(* Logix 5000 project; controller reports 1756-L63 rev 20.11; software revision 20.04; part 5 of 52 *)

        [413].time.Second := 59, [414].log_data[0].min := 1.0, [414].log_data[0].max := 1.0, [414].log_data[0].total := 900.0, [414].log_data[0].time := 900.0, [414].log_data[0].minminute := 45, [414].log_data[0].maxminute := 45, [414].log_data[0].valid := 1, [414].log_data[1].valid := 1, [414].log_data[2].valid := 1, [414].log_data[3].valid := 1, [414].log_data[4].valid := 1, [414].log_data[5].valid := 1, [414].log_data[6].valid := 1, [414].log_data[7].valid := 1, [414].log_data[8].valid := 1, [414].log_data[9].valid := 1, [414].log_data[10].valid := 1, [414].log_data[11].valid := 1, [414].log_data[12].valid := 1, [414].log_data[13].valid := 1, [414].log_data[14].valid := 1, [414].log_data[15].valid := 1, [414].log_data[16].valid := 1, [414].log_data[17].valid := 1, [414].log_data[18].valid := 1, [414].log_data[19].valid := 1, [414].time.Year := 2023, [414].time.Month := 1, [414].time.Day := 11, [414].time.Hour := 23, [414].time.Minute := 59, [414].time.Second := 59, [415].log_data[0].min := 1.0, [415].log_data[0].max := 1.0, [415].log_data[0].total := 900.0, [415].log_data[0].time := 900.0, [415].log_data[0].valid := 1, [415].log_data[1].valid := 1, [415].log_data[2].valid := 1, [415].log_data[3].valid := 1, [415].log_data[4].valid := 1, [415].log_data[5].valid := 1, [415].log_data[6].valid := 1, [415].log_data[7].valid := 1, [415].log_data[8].valid := 1, [415].log_data[9].valid := 1, [415].log_data[10].valid := 1, [415].log_data[11].valid := 1, [415].log_data[12].valid := 1, [415].log_data[13].valid := 1, [415].log_data[14].valid := 1, [415].log_data[15].valid := 1, [415].log_data[16].valid := 1, [415].log_data[17].valid := 1, [415].log_data[18].valid := 1, [415].log_data[19].valid := 1, [415].time.Year := 2023, [415].time.Month := 1, [415].time.Day := 12,
        [415].time.Minute := 14, [415].time.Second := 59, [416].log_data[0].min := 1.0, [416].log_data[0].max := 1.0, [416].log_data[0].total := 900.0, [416].log_data[0].time := 900.0, [416].log_data[0].minminute := 15, [416].log_data[0].maxminute := 15, [416].log_data[0].valid := 1, [416].log_data[1].valid := 1, [416].log_data[2].valid := 1, [416].log_data[3].valid := 1, [416].log_data[4].valid := 1, [416].log_data[5].valid := 1, [416].log_data[6].valid := 1, [416].log_data[7].valid := 1, [416].log_data[8].valid := 1, [416].log_data[9].valid := 1, [416].log_data[10].valid := 1, [416].log_data[11].valid := 1, [416].log_data[12].valid := 1, [416].log_data[13].valid := 1, [416].log_data[14].valid := 1, [416].log_data[15].valid := 1, [416].log_data[16].valid := 1, [416].log_data[17].valid := 1, [416].log_data[18].valid := 1, [416].log_data[19].valid := 1, [416].time.Year := 2023, [416].time.Month := 1, [416].time.Day := 12, [416].time.Minute := 29, [416].time.Second := 59, [417].log_data[0].min := 1.0, [417].log_data[0].max := 1.0, [417].log_data[0].total := 900.0, [417].log_data[0].time := 900.0, [417].log_data[0].minminute := 30, [417].log_data[0].maxminute := 30, [417].log_data[0].valid := 1, [417].log_data[1].valid := 1, [417].log_data[2].valid := 1, [417].log_data[3].valid := 1, [417].log_data[4].valid := 1, [417].log_data[5].valid := 1, [417].log_data[6].valid := 1, [417].log_data[7].valid := 1, [417].log_data[8].valid := 1, [417].log_data[9].valid := 1, [417].log_data[10].valid := 1, [417].log_data[11].valid := 1, [417].log_data[12].valid := 1, [417].log_data[13].valid := 1, [417].log_data[14].valid := 1, [417].log_data[15].valid := 1, [417].log_data[16].valid := 1, [417].log_data[17].valid := 1, [417].log_data[18].valid := 1, [417].log_data[19].valid := 1, [417].time.Year := 2023,
        [417].time.Month := 1, [417].time.Day := 12, [417].time.Minute := 44, [417].time.Second := 59, [418].log_data[0].min := 1.0, [418].log_data[0].max := 1.0, [418].log_data[0].total := 900.0, [418].log_data[0].time := 900.0, [418].log_data[0].minminute := 45, [418].log_data[0].maxminute := 45, [418].log_data[0].valid := 1, [418].log_data[1].valid := 1, [418].log_data[2].valid := 1, [418].log_data[3].valid := 1, [418].log_data[4].valid := 1, [418].log_data[5].valid := 1, [418].log_data[6].valid := 1, [418].log_data[7].valid := 1, [418].log_data[8].valid := 1, [418].log_data[9].valid := 1, [418].log_data[10].valid := 1, [418].log_data[11].valid := 1, [418].log_data[12].valid := 1, [418].log_data[13].valid := 1, [418].log_data[14].valid := 1, [418].log_data[15].valid := 1, [418].log_data[16].valid := 1, [418].log_data[17].valid := 1, [418].log_data[18].valid := 1, [418].log_data[19].valid := 1, [418].time.Year := 2023, [418].time.Month := 1, [418].time.Day := 12, [418].time.Minute := 59, [418].time.Second := 59, [419].log_data[0].min := 1.0, [419].log_data[0].max := 1.0, [419].log_data[0].total := 899.5, [419].log_data[0].time := 899.5, [419].log_data[0].valid := 1, [419].log_data[1].valid := 1, [419].log_data[2].valid := 1, [419].log_data[3].valid := 1, [419].log_data[4].valid := 1, [419].log_data[5].valid := 1, [419].log_data[6].valid := 1, [419].log_data[7].valid := 1, [419].log_data[8].valid := 1, [419].log_data[9].valid := 1, [419].log_data[10].valid := 1, [419].log_data[11].valid := 1, [419].log_data[12].valid := 1, [419].log_data[13].valid := 1, [419].log_data[14].valid := 1, [419].log_data[15].valid := 1, [419].log_data[16].valid := 1, [419].log_data[17].valid := 1, [419].log_data[18].valid := 1, [419].log_data[19].valid := 1, [419].time.Year := 2023,
        [419].time.Month := 1, [419].time.Day := 12, [419].time.Hour := 1, [419].time.Minute := 14, [419].time.Second := 59, [420].log_data[0].min := 1.0, [420].log_data[0].max := 1.0, [420].log_data[0].total := 900.0, [420].log_data[0].time := 900.0, [420].log_data[0].minminute := 15, [420].log_data[0].maxminute := 15, [420].log_data[0].valid := 1, [420].log_data[1].valid := 1, [420].log_data[2].valid := 1, [420].log_data[3].valid := 1, [420].log_data[4].valid := 1, [420].log_data[5].valid := 1, [420].log_data[6].valid := 1, [420].log_data[7].valid := 1, [420].log_data[8].valid := 1, [420].log_data[9].valid := 1, [420].log_data[10].valid := 1, [420].log_data[11].valid := 1, [420].log_data[12].valid := 1, [420].log_data[13].valid := 1, [420].log_data[14].valid := 1, [420].log_data[15].valid := 1, [420].log_data[16].valid := 1, [420].log_data[17].valid := 1, [420].log_data[18].valid := 1, [420].log_data[19].valid := 1, [420].time.Year := 2023, [420].time.Month := 1, [420].time.Day := 12, [420].time.Hour := 1, [420].time.Minute := 29, [420].time.Second := 59, [421].log_data[0].min := 1.0, [421].log_data[0].max := 1.0, [421].log_data[0].total := 900.0, [421].log_data[0].time := 900.0, [421].log_data[0].minminute := 30, [421].log_data[0].maxminute := 30, [421].log_data[0].valid := 1, [421].log_data[1].valid := 1, [421].log_data[2].valid := 1, [421].log_data[3].valid := 1, [421].log_data[4].valid := 1, [421].log_data[5].valid := 1, [421].log_data[6].valid := 1, [421].log_data[7].valid := 1, [421].log_data[8].valid := 1, [421].log_data[9].valid := 1, [421].log_data[10].valid := 1, [421].log_data[11].valid := 1, [421].log_data[12].valid := 1, [421].log_data[13].valid := 1, [421].log_data[14].valid := 1, [421].log_data[15].valid := 1, [421].log_data[16].valid := 1,
        [421].log_data[17].valid := 1, [421].log_data[18].valid := 1, [421].log_data[19].valid := 1, [421].time.Year := 2023, [421].time.Month := 1, [421].time.Day := 12, [421].time.Hour := 1, [421].time.Minute := 44, [421].time.Second := 59, [422].log_data[0].min := 1.0, [422].log_data[0].max := 1.0, [422].log_data[0].total := 900.0, [422].log_data[0].time := 900.0, [422].log_data[0].minminute := 45, [422].log_data[0].maxminute := 45, [422].log_data[0].valid := 1, [422].log_data[1].valid := 1, [422].log_data[2].valid := 1, [422].log_data[3].valid := 1, [422].log_data[4].valid := 1, [422].log_data[5].valid := 1, [422].log_data[6].valid := 1, [422].log_data[7].valid := 1, [422].log_data[8].valid := 1, [422].log_data[9].valid := 1, [422].log_data[10].valid := 1, [422].log_data[11].valid := 1, [422].log_data[12].valid := 1, [422].log_data[13].valid := 1, [422].log_data[14].valid := 1, [422].log_data[15].valid := 1, [422].log_data[16].valid := 1, [422].log_data[17].valid := 1, [422].log_data[18].valid := 1, [422].log_data[19].valid := 1, [422].time.Year := 2023, [422].time.Month := 1, [422].time.Day := 12, [422].time.Hour := 1, [422].time.Minute := 59, [422].time.Second := 59, [423].log_data[0].min := 1.0, [423].log_data[0].max := 1.0, [423].log_data[0].total := 900.0, [423].log_data[0].time := 900.0, [423].log_data[0].valid := 1, [423].log_data[1].valid := 1, [423].log_data[2].valid := 1, [423].log_data[3].valid := 1, [423].log_data[4].valid := 1, [423].log_data[5].valid := 1, [423].log_data[6].valid := 1, [423].log_data[7].valid := 1, [423].log_data[8].valid := 1, [423].log_data[9].valid := 1, [423].log_data[10].valid := 1, [423].log_data[11].valid := 1, [423].log_data[12].valid := 1, [423].log_data[13].valid := 1, [423].log_data[14].valid := 1,
        [423].log_data[15].valid := 1, [423].log_data[16].valid := 1, [423].log_data[17].valid := 1, [423].log_data[18].valid := 1, [423].log_data[19].valid := 1, [423].time.Year := 2023, [423].time.Month := 1, [423].time.Day := 12, [423].time.Hour := 2, [423].time.Minute := 14, [423].time.Second := 59, [424].log_data[0].min := 1.0, [424].log_data[0].max := 1.0, [424].log_data[0].total := 900.0, [424].log_data[0].time := 900.0, [424].log_data[0].minminute := 15, [424].log_data[0].maxminute := 15, [424].log_data[0].valid := 1, [424].log_data[1].valid := 1, [424].log_data[2].valid := 1, [424].log_data[3].valid := 1, [424].log_data[4].valid := 1, [424].log_data[5].valid := 1, [424].log_data[6].valid := 1, [424].log_data[7].valid := 1, [424].log_data[8].valid := 1, [424].log_data[9].valid := 1, [424].log_data[10].valid := 1, [424].log_data[11].valid := 1, [424].log_data[12].valid := 1, [424].log_data[13].valid := 1, [424].log_data[14].valid := 1, [424].log_data[15].valid := 1, [424].log_data[16].valid := 1, [424].log_data[17].valid := 1, [424].log_data[18].valid := 1, [424].log_data[19].valid := 1, [424].time.Year := 2023, [424].time.Month := 1, [424].time.Day := 12, [424].time.Hour := 2, [424].time.Minute := 29, [424].time.Second := 59, [425].log_data[0].min := 1.0, [425].log_data[0].max := 1.0, [425].log_data[0].total := 900.0, [425].log_data[0].time := 900.0, [425].log_data[0].minminute := 30, [425].log_data[0].maxminute := 30, [425].log_data[0].valid := 1, [425].log_data[1].valid := 1, [425].log_data[2].valid := 1, [425].log_data[3].valid := 1, [425].log_data[4].valid := 1, [425].log_data[5].valid := 1, [425].log_data[6].valid := 1, [425].log_data[7].valid := 1, [425].log_data[8].valid := 1, [425].log_data[9].valid := 1, [425].log_data[10].valid := 1,
        [425].log_data[11].valid := 1, [425].log_data[12].valid := 1, [425].log_data[13].valid := 1, [425].log_data[14].valid := 1, [425].log_data[15].valid := 1, [425].log_data[16].valid := 1, [425].log_data[17].valid := 1, [425].log_data[18].valid := 1, [425].log_data[19].valid := 1, [425].time.Year := 2023, [425].time.Month := 1, [425].time.Day := 12, [425].time.Hour := 2, [425].time.Minute := 44, [425].time.Second := 59, [426].log_data[0].min := 1.0, [426].log_data[0].max := 1.0, [426].log_data[0].total := 900.0, [426].log_data[0].time := 900.0, [426].log_data[0].minminute := 45, [426].log_data[0].maxminute := 45, [426].log_data[0].valid := 1, [426].log_data[1].valid := 1, [426].log_data[2].valid := 1, [426].log_data[3].valid := 1, [426].log_data[4].valid := 1, [426].log_data[5].valid := 1, [426].log_data[6].valid := 1, [426].log_data[7].valid := 1, [426].log_data[8].valid := 1, [426].log_data[9].valid := 1, [426].log_data[10].valid := 1, [426].log_data[11].valid := 1, [426].log_data[12].valid := 1, [426].log_data[13].valid := 1, [426].log_data[14].valid := 1, [426].log_data[15].valid := 1, [426].log_data[16].valid := 1, [426].log_data[17].valid := 1, [426].log_data[18].valid := 1, [426].log_data[19].valid := 1, [426].time.Year := 2023, [426].time.Month := 1, [426].time.Day := 12, [426].time.Hour := 2, [426].time.Minute := 59, [426].time.Second := 59, [427].log_data[0].min := 1.0, [427].log_data[0].max := 1.0, [427].log_data[0].total := 900.0, [427].log_data[0].time := 900.0, [427].log_data[0].valid := 1, [427].log_data[1].valid := 1, [427].log_data[2].valid := 1, [427].log_data[3].valid := 1, [427].log_data[4].valid := 1, [427].log_data[5].valid := 1, [427].log_data[6].valid := 1, [427].log_data[7].valid := 1, [427].log_data[8].valid := 1,
        [427].log_data[9].valid := 1, [427].log_data[10].valid := 1, [427].log_data[11].valid := 1, [427].log_data[12].valid := 1, [427].log_data[13].valid := 1, [427].log_data[14].valid := 1, [427].log_data[15].valid := 1, [427].log_data[16].valid := 1, [427].log_data[17].valid := 1, [427].log_data[18].valid := 1, [427].log_data[19].valid := 1, [427].time.Year := 2023, [427].time.Month := 1, [427].time.Day := 12, [427].time.Hour := 3, [427].time.Minute := 14, [427].time.Second := 59, [428].log_data[0].min := 1.0, [428].log_data[0].max := 1.0, [428].log_data[0].total := 900.0, [428].log_data[0].time := 900.0, [428].log_data[0].minminute := 15, [428].log_data[0].maxminute := 15, [428].log_data[0].valid := 1, [428].log_data[1].valid := 1, [428].log_data[2].valid := 1, [428].log_data[3].valid := 1, [428].log_data[4].valid := 1, [428].log_data[5].valid := 1, [428].log_data[6].valid := 1, [428].log_data[7].valid := 1, [428].log_data[8].valid := 1, [428].log_data[9].valid := 1, [428].log_data[10].valid := 1, [428].log_data[11].valid := 1, [428].log_data[12].valid := 1, [428].log_data[13].valid := 1, [428].log_data[14].valid := 1, [428].log_data[15].valid := 1, [428].log_data[16].valid := 1, [428].log_data[17].valid := 1, [428].log_data[18].valid := 1, [428].log_data[19].valid := 1, [428].time.Year := 2023, [428].time.Month := 1, [428].time.Day := 12, [428].time.Hour := 3, [428].time.Minute := 29, [428].time.Second := 59, [429].log_data[0].min := 1.0, [429].log_data[0].max := 1.0, [429].log_data[0].total := 900.0, [429].log_data[0].time := 900.0, [429].log_data[0].minminute := 30, [429].log_data[0].maxminute := 30, [429].log_data[0].valid := 1, [429].log_data[1].valid := 1, [429].log_data[2].valid := 1, [429].log_data[3].valid := 1, [429].log_data[4].valid := 1,
        [429].log_data[5].valid := 1, [429].log_data[6].valid := 1, [429].log_data[7].valid := 1, [429].log_data[8].valid := 1, [429].log_data[9].valid := 1, [429].log_data[10].valid := 1, [429].log_data[11].valid := 1, [429].log_data[12].valid := 1, [429].log_data[13].valid := 1, [429].log_data[14].valid := 1, [429].log_data[15].valid := 1, [429].log_data[16].valid := 1, [429].log_data[17].valid := 1, [429].log_data[18].valid := 1, [429].log_data[19].valid := 1, [429].time.Year := 2023, [429].time.Month := 1, [429].time.Day := 12, [429].time.Hour := 3, [429].time.Minute := 44, [429].time.Second := 59, [430].log_data[0].min := 1.0, [430].log_data[0].max := 1.0, [430].log_data[0].total := 900.0, [430].log_data[0].time := 900.0, [430].log_data[0].minminute := 45, [430].log_data[0].maxminute := 45, [430].log_data[0].valid := 1, [430].log_data[1].valid := 1, [430].log_data[2].valid := 1, [430].log_data[3].valid := 1, [430].log_data[4].valid := 1, [430].log_data[5].valid := 1, [430].log_data[6].valid := 1, [430].log_data[7].valid := 1, [430].log_data[8].valid := 1, [430].log_data[9].valid := 1, [430].log_data[10].valid := 1, [430].log_data[11].valid := 1, [430].log_data[12].valid := 1, [430].log_data[13].valid := 1, [430].log_data[14].valid := 1, [430].log_data[15].valid := 1, [430].log_data[16].valid := 1, [430].log_data[17].valid := 1, [430].log_data[18].valid := 1, [430].log_data[19].valid := 1, [430].time.Year := 2023, [430].time.Month := 1, [430].time.Day := 12, [430].time.Hour := 3, [430].time.Minute := 59, [430].time.Second := 59, [431].log_data[0].min := 1.0, [431].log_data[0].max := 1.0, [431].log_data[0].total := 900.0, [431].log_data[0].time := 900.0, [431].log_data[0].valid := 1, [431].log_data[1].valid := 1, [431].log_data[2].valid := 1,
        [431].log_data[3].valid := 1, [431].log_data[4].valid := 1, [431].log_data[5].valid := 1, [431].log_data[6].valid := 1, [431].log_data[7].valid := 1, [431].log_data[8].valid := 1, [431].log_data[9].valid := 1, [431].log_data[10].valid := 1, [431].log_data[11].valid := 1, [431].log_data[12].valid := 1, [431].log_data[13].valid := 1, [431].log_data[14].valid := 1, [431].log_data[15].valid := 1, [431].log_data[16].valid := 1, [431].log_data[17].valid := 1, [431].log_data[18].valid := 1, [431].log_data[19].valid := 1, [431].time.Year := 2023, [431].time.Month := 1, [431].time.Day := 12, [431].time.Hour := 4, [431].time.Minute := 14, [431].time.Second := 59, [432].log_data[0].min := 1.0, [432].log_data[0].max := 1.0, [432].log_data[0].total := 900.0, [432].log_data[0].time := 900.0, [432].log_data[0].minminute := 15, [432].log_data[0].maxminute := 15, [432].log_data[0].valid := 1, [432].log_data[1].valid := 1, [432].log_data[2].valid := 1, [432].log_data[3].valid := 1, [432].log_data[4].valid := 1, [432].log_data[5].valid := 1, [432].log_data[6].valid := 1, [432].log_data[7].valid := 1, [432].log_data[8].valid := 1, [432].log_data[9].valid := 1, [432].log_data[10].valid := 1, [432].log_data[11].valid := 1, [432].log_data[12].valid := 1, [432].log_data[13].valid := 1, [432].log_data[14].valid := 1, [432].log_data[15].valid := 1, [432].log_data[16].valid := 1, [432].log_data[17].valid := 1, [432].log_data[18].valid := 1, [432].log_data[19].valid := 1, [432].time.Year := 2023, [432].time.Month := 1, [432].time.Day := 12, [432].time.Hour := 4, [432].time.Minute := 29, [432].time.Second := 59, [433].log_data[0].min := 1.0, [433].log_data[0].max := 1.0, [433].log_data[0].total := 900.0, [433].log_data[0].time := 900.0, [433].log_data[0].minminute := 30,
        [433].log_data[0].maxminute := 30, [433].log_data[0].valid := 1, [433].log_data[1].valid := 1, [433].log_data[2].valid := 1, [433].log_data[3].valid := 1, [433].log_data[4].valid := 1, [433].log_data[5].valid := 1, [433].log_data[6].valid := 1, [433].log_data[7].valid := 1, [433].log_data[8].valid := 1, [433].log_data[9].valid := 1, [433].log_data[10].valid := 1, [433].log_data[11].valid := 1, [433].log_data[12].valid := 1, [433].log_data[13].valid := 1, [433].log_data[14].valid := 1, [433].log_data[15].valid := 1, [433].log_data[16].valid := 1, [433].log_data[17].valid := 1, [433].log_data[18].valid := 1, [433].log_data[19].valid := 1, [433].time.Year := 2023, [433].time.Month := 1, [433].time.Day := 12, [433].time.Hour := 4, [433].time.Minute := 44, [433].time.Second := 59, [434].log_data[0].min := 1.0, [434].log_data[0].max := 1.0, [434].log_data[0].total := 900.0, [434].log_data[0].time := 900.0, [434].log_data[0].minminute := 45, [434].log_data[0].maxminute := 45, [434].log_data[0].valid := 1, [434].log_data[1].valid := 1, [434].log_data[2].valid := 1, [434].log_data[3].valid := 1, [434].log_data[4].valid := 1, [434].log_data[5].valid := 1, [434].log_data[6].valid := 1, [434].log_data[7].valid := 1, [434].log_data[8].valid := 1, [434].log_data[9].valid := 1, [434].log_data[10].valid := 1, [434].log_data[11].valid := 1, [434].log_data[12].valid := 1, [434].log_data[13].valid := 1, [434].log_data[14].valid := 1, [434].log_data[15].valid := 1, [434].log_data[16].valid := 1, [434].log_data[17].valid := 1, [434].log_data[18].valid := 1, [434].log_data[19].valid := 1, [434].time.Year := 2023, [434].time.Month := 1, [434].time.Day := 12, [434].time.Hour := 4, [434].time.Minute := 59, [434].time.Second := 59, [435].log_data[0].min := 1.0,
        [435].log_data[0].max := 1.0, [435].log_data[0].total := 900.0, [435].log_data[0].time := 900.0, [435].log_data[0].valid := 1, [435].log_data[1].valid := 1, [435].log_data[2].valid := 1, [435].log_data[3].valid := 1, [435].log_data[4].valid := 1, [435].log_data[5].valid := 1, [435].log_data[6].valid := 1, [435].log_data[7].valid := 1, [435].log_data[8].valid := 1, [435].log_data[9].valid := 1, [435].log_data[10].valid := 1, [435].log_data[11].valid := 1, [435].log_data[12].valid := 1, [435].log_data[13].valid := 1, [435].log_data[14].valid := 1, [435].log_data[15].valid := 1, [435].log_data[16].valid := 1, [435].log_data[17].valid := 1, [435].log_data[18].valid := 1, [435].log_data[19].valid := 1, [435].time.Year := 2023, [435].time.Month := 1, [435].time.Day := 12, [435].time.Hour := 5, [435].time.Minute := 14, [435].time.Second := 59, [436].log_data[0].min := 1.0, [436].log_data[0].max := 1.0, [436].log_data[0].total := 900.0, [436].log_data[0].time := 900.0, [436].log_data[0].minminute := 15, [436].log_data[0].maxminute := 15, [436].log_data[0].valid := 1, [436].log_data[1].valid := 1, [436].log_data[2].valid := 1, [436].log_data[3].valid := 1, [436].log_data[4].valid := 1, [436].log_data[5].valid := 1, [436].log_data[6].valid := 1, [436].log_data[7].valid := 1, [436].log_data[8].valid := 1, [436].log_data[9].valid := 1, [436].log_data[10].valid := 1, [436].log_data[11].valid := 1, [436].log_data[12].valid := 1, [436].log_data[13].valid := 1, [436].log_data[14].valid := 1, [436].log_data[15].valid := 1, [436].log_data[16].valid := 1, [436].log_data[17].valid := 1, [436].log_data[18].valid := 1, [436].log_data[19].valid := 1, [436].time.Year := 2023, [436].time.Month := 1, [436].time.Day := 12, [436].time.Hour := 5, [436].time.Minute := 29,
        [436].time.Second := 59, [437].log_data[0].min := 1.0, [437].log_data[0].max := 1.0, [437].log_data[0].total := 900.0, [437].log_data[0].time := 900.0, [437].log_data[0].minminute := 30, [437].log_data[0].maxminute := 30, [437].log_data[0].valid := 1, [437].log_data[1].valid := 1, [437].log_data[2].valid := 1, [437].log_data[3].valid := 1, [437].log_data[4].valid := 1, [437].log_data[5].valid := 1, [437].log_data[6].valid := 1, [437].log_data[7].valid := 1, [437].log_data[8].valid := 1, [437].log_data[9].valid := 1, [437].log_data[10].valid := 1, [437].log_data[11].valid := 1, [437].log_data[12].valid := 1, [437].log_data[13].valid := 1, [437].log_data[14].valid := 1, [437].log_data[15].valid := 1, [437].log_data[16].valid := 1, [437].log_data[17].valid := 1, [437].log_data[18].valid := 1, [437].log_data[19].valid := 1, [437].time.Year := 2023, [437].time.Month := 1, [437].time.Day := 12, [437].time.Hour := 5, [437].time.Minute := 44, [437].time.Second := 59, [438].log_data[0].min := 1.0, [438].log_data[0].max := 1.0, [438].log_data[0].total := 900.0, [438].log_data[0].time := 900.0, [438].log_data[0].minminute := 45, [438].log_data[0].maxminute := 45, [438].log_data[0].valid := 1, [438].log_data[1].valid := 1, [438].log_data[2].valid := 1, [438].log_data[3].valid := 1, [438].log_data[4].valid := 1, [438].log_data[5].valid := 1, [438].log_data[6].valid := 1, [438].log_data[7].valid := 1, [438].log_data[8].valid := 1, [438].log_data[9].valid := 1, [438].log_data[10].valid := 1, [438].log_data[11].valid := 1, [438].log_data[12].valid := 1, [438].log_data[13].valid := 1, [438].log_data[14].valid := 1, [438].log_data[15].valid := 1, [438].log_data[16].valid := 1, [438].log_data[17].valid := 1, [438].log_data[18].valid := 1, [438].log_data[19].valid := 1, [438].time.Year := 2023,
        [438].time.Month := 1, [438].time.Day := 12, [438].time.Hour := 5, [438].time.Minute := 59, [438].time.Second := 59, [439].log_data[0].min := 1.0, [439].log_data[0].max := 1.0, [439].log_data[0].total := 900.0, [439].log_data[0].time := 900.0, [439].log_data[0].valid := 1, [439].log_data[1].valid := 1, [439].log_data[2].valid := 1, [439].log_data[3].valid := 1, [439].log_data[4].valid := 1, [439].log_data[5].valid := 1, [439].log_data[6].valid := 1, [439].log_data[7].valid := 1, [439].log_data[8].valid := 1, [439].log_data[9].valid := 1, [439].log_data[10].valid := 1, [439].log_data[11].valid := 1, [439].log_data[12].valid := 1, [439].log_data[13].valid := 1, [439].log_data[14].valid := 1, [439].log_data[15].valid := 1, [439].log_data[16].valid := 1, [439].log_data[17].valid := 1, [439].log_data[18].valid := 1, [439].log_data[19].valid := 1, [439].time.Year := 2023, [439].time.Month := 1, [439].time.Day := 12, [439].time.Hour := 6, [439].time.Minute := 14, [439].time.Second := 59, [440].log_data[0].min := 1.0, [440].log_data[0].max := 1.0, [440].log_data[0].total := 900.0, [440].log_data[0].time := 900.0, [440].log_data[0].minminute := 15, [440].log_data[0].maxminute := 15, [440].log_data[0].valid := 1, [440].log_data[1].valid := 1, [440].log_data[2].valid := 1, [440].log_data[3].valid := 1, [440].log_data[4].valid := 1, [440].log_data[5].valid := 1, [440].log_data[6].valid := 1, [440].log_data[7].valid := 1, [440].log_data[8].valid := 1, [440].log_data[9].valid := 1, [440].log_data[10].valid := 1, [440].log_data[11].valid := 1, [440].log_data[12].valid := 1, [440].log_data[13].valid := 1, [440].log_data[14].valid := 1, [440].log_data[15].valid := 1, [440].log_data[16].valid := 1, [440].log_data[17].valid := 1, [440].log_data[18].valid := 1,
        [440].log_data[19].valid := 1, [440].time.Year := 2023, [440].time.Month := 1, [440].time.Day := 12, [440].time.Hour := 6, [440].time.Minute := 29, [440].time.Second := 59, [441].log_data[0].min := 1.0, [441].log_data[0].max := 1.0, [441].log_data[0].total := 900.0, [441].log_data[0].time := 900.0, [441].log_data[0].minminute := 30, [441].log_data[0].maxminute := 30, [441].log_data[0].valid := 1, [441].log_data[1].valid := 1, [441].log_data[2].valid := 1, [441].log_data[3].valid := 1, [441].log_data[4].valid := 1, [441].log_data[5].valid := 1, [441].log_data[6].valid := 1, [441].log_data[7].valid := 1, [441].log_data[8].valid := 1, [441].log_data[9].valid := 1, [441].log_data[10].valid := 1, [441].log_data[11].valid := 1, [441].log_data[12].valid := 1, [441].log_data[13].valid := 1, [441].log_data[14].valid := 1, [441].log_data[15].valid := 1, [441].log_data[16].valid := 1, [441].log_data[17].valid := 1, [441].log_data[18].valid := 1, [441].log_data[19].valid := 1, [441].time.Year := 2023, [441].time.Month := 1, [441].time.Day := 12, [441].time.Hour := 6, [441].time.Minute := 44, [441].time.Second := 59, [442].log_data[0].min := 1.0, [442].log_data[0].max := 1.0, [442].log_data[0].total := 900.0, [442].log_data[0].time := 900.0, [442].log_data[0].minminute := 45, [442].log_data[0].maxminute := 45, [442].log_data[0].valid := 1, [442].log_data[1].valid := 1, [442].log_data[2].valid := 1, [442].log_data[3].valid := 1, [442].log_data[4].valid := 1, [442].log_data[5].valid := 1, [442].log_data[6].valid := 1, [442].log_data[7].valid := 1, [442].log_data[8].valid := 1, [442].log_data[9].valid := 1, [442].log_data[10].valid := 1, [442].log_data[11].valid := 1, [442].log_data[12].valid := 1, [442].log_data[13].valid := 1, [442].log_data[14].valid := 1,
        [442].log_data[15].valid := 1, [442].log_data[16].valid := 1, [442].log_data[17].valid := 1, [442].log_data[18].valid := 1, [442].log_data[19].valid := 1, [442].time.Year := 2023, [442].time.Month := 1, [442].time.Day := 12, [442].time.Hour := 6, [442].time.Minute := 59, [442].time.Second := 59, [443].log_data[0].min := 1.0, [443].log_data[0].max := 1.0, [443].log_data[0].total := 900.0, [443].log_data[0].time := 900.0, [443].log_data[0].valid := 1, [443].log_data[1].valid := 1, [443].log_data[2].valid := 1, [443].log_data[3].valid := 1, [443].log_data[4].valid := 1, [443].log_data[5].valid := 1, [443].log_data[6].valid := 1, [443].log_data[7].valid := 1, [443].log_data[8].valid := 1, [443].log_data[9].valid := 1, [443].log_data[10].valid := 1, [443].log_data[11].valid := 1, [443].log_data[12].valid := 1, [443].log_data[13].valid := 1, [443].log_data[14].valid := 1, [443].log_data[15].valid := 1, [443].log_data[16].valid := 1, [443].log_data[17].valid := 1, [443].log_data[18].valid := 1, [443].log_data[19].valid := 1, [443].time.Year := 2023, [443].time.Month := 1, [443].time.Day := 12, [443].time.Hour := 7, [443].time.Minute := 14, [443].time.Second := 59, [444].log_data[0].min := 1.0, [444].log_data[0].max := 1.0, [444].log_data[0].total := 900.0, [444].log_data[0].time := 900.0, [444].log_data[0].minminute := 15, [444].log_data[0].maxminute := 15, [444].log_data[0].valid := 1, [444].log_data[1].valid := 1, [444].log_data[2].valid := 1, [444].log_data[3].valid := 1, [444].log_data[4].valid := 1, [444].log_data[5].valid := 1, [444].log_data[6].valid := 1, [444].log_data[7].valid := 1, [444].log_data[8].valid := 1, [444].log_data[9].valid := 1, [444].log_data[10].valid := 1, [444].log_data[11].valid := 1, [444].log_data[12].valid := 1,
        [444].log_data[13].valid := 1, [444].log_data[14].valid := 1, [444].log_data[15].valid := 1, [444].log_data[16].valid := 1, [444].log_data[17].valid := 1, [444].log_data[18].valid := 1, [444].log_data[19].valid := 1, [444].time.Year := 2023, [444].time.Month := 1, [444].time.Day := 12, [444].time.Hour := 7, [444].time.Minute := 29, [444].time.Second := 59, [445].log_data[0].min := 1.0, [445].log_data[0].max := 1.0, [445].log_data[0].total := 900.0, [445].log_data[0].time := 900.0, [445].log_data[0].minminute := 30, [445].log_data[0].maxminute := 30, [445].log_data[0].valid := 1, [445].log_data[1].valid := 1, [445].log_data[2].valid := 1, [445].log_data[3].valid := 1, [445].log_data[4].valid := 1, [445].log_data[5].valid := 1, [445].log_data[6].valid := 1, [445].log_data[7].valid := 1, [445].log_data[8].valid := 1, [445].log_data[9].valid := 1, [445].log_data[10].valid := 1, [445].log_data[11].valid := 1, [445].log_data[12].valid := 1, [445].log_data[13].valid := 1, [445].log_data[14].valid := 1, [445].log_data[15].valid := 1, [445].log_data[16].valid := 1, [445].log_data[17].valid := 1, [445].log_data[18].valid := 1, [445].log_data[19].valid := 1, [445].time.Year := 2023, [445].time.Month := 1, [445].time.Day := 12, [445].time.Hour := 7, [445].time.Minute := 44, [445].time.Second := 59, [446].log_data[0].min := 1.0, [446].log_data[0].max := 1.0, [446].log_data[0].total := 900.0, [446].log_data[0].time := 900.0, [446].log_data[0].minminute := 45, [446].log_data[0].maxminute := 45, [446].log_data[0].valid := 1, [446].log_data[1].valid := 1, [446].log_data[2].valid := 1, [446].log_data[3].valid := 1, [446].log_data[4].valid := 1, [446].log_data[5].valid := 1, [446].log_data[6].valid := 1, [446].log_data[7].valid := 1, [446].log_data[8].valid := 1,
        [446].log_data[9].valid := 1, [446].log_data[10].valid := 1, [446].log_data[11].valid := 1, [446].log_data[12].valid := 1, [446].log_data[13].valid := 1, [446].log_data[14].valid := 1, [446].log_data[15].valid := 1, [446].log_data[16].valid := 1, [446].log_data[17].valid := 1, [446].log_data[18].valid := 1, [446].log_data[19].valid := 1, [446].time.Year := 2023, [446].time.Month := 1, [446].time.Day := 12, [446].time.Hour := 7, [446].time.Minute := 59, [446].time.Second := 59, [447].log_data[0].min := 1.0, [447].log_data[0].max := 1.0, [447].log_data[0].total := 900.0, [447].log_data[0].time := 900.0, [447].log_data[0].valid := 1, [447].log_data[1].valid := 1, [447].log_data[2].valid := 1, [447].log_data[3].valid := 1, [447].log_data[4].valid := 1, [447].log_data[5].valid := 1, [447].log_data[6].valid := 1, [447].log_data[7].valid := 1, [447].log_data[8].valid := 1, [447].log_data[9].valid := 1, [447].log_data[10].valid := 1, [447].log_data[11].valid := 1, [447].log_data[12].valid := 1, [447].log_data[13].valid := 1, [447].log_data[14].valid := 1, [447].log_data[15].valid := 1, [447].log_data[16].valid := 1, [447].log_data[17].valid := 1, [447].log_data[18].valid := 1, [447].log_data[19].valid := 1, [447].time.Year := 2023, [447].time.Month := 1, [447].time.Day := 12, [447].time.Hour := 8, [447].time.Minute := 14, [447].time.Second := 59, [448].log_data[0].min := 1.0, [448].log_data[0].max := 1.0, [448].log_data[0].total := 900.0, [448].log_data[0].time := 900.0, [448].log_data[0].minminute := 15, [448].log_data[0].maxminute := 15, [448].log_data[0].valid := 1, [448].log_data[1].valid := 1, [448].log_data[2].valid := 1, [448].log_data[3].valid := 1, [448].log_data[4].valid := 1, [448].log_data[5].valid := 1, [448].log_data[6].valid := 1,
        [448].log_data[7].valid := 1, [448].log_data[8].valid := 1, [448].log_data[9].valid := 1, [448].log_data[10].valid := 1, [448].log_data[11].valid := 1, [448].log_data[12].valid := 1, [448].log_data[13].valid := 1, [448].log_data[14].valid := 1, [448].log_data[15].valid := 1, [448].log_data[16].valid := 1, [448].log_data[17].valid := 1, [448].log_data[18].valid := 1, [448].log_data[19].valid := 1, [448].time.Year := 2023, [448].time.Month := 1, [448].time.Day := 12, [448].time.Hour := 8, [448].time.Minute := 29, [448].time.Second := 59, [449].log_data[0].min := 1.0, [449].log_data[0].max := 1.0, [449].log_data[0].total := 900.0, [449].log_data[0].time := 900.0, [449].log_data[0].minminute := 30, [449].log_data[0].maxminute := 30, [449].log_data[0].valid := 1, [449].log_data[1].valid := 1, [449].log_data[2].valid := 1, [449].log_data[3].valid := 1, [449].log_data[4].valid := 1, [449].log_data[5].valid := 1, [449].log_data[6].valid := 1, [449].log_data[7].valid := 1, [449].log_data[8].valid := 1, [449].log_data[9].valid := 1, [449].log_data[10].valid := 1, [449].log_data[11].valid := 1, [449].log_data[12].valid := 1, [449].log_data[13].valid := 1, [449].log_data[14].valid := 1, [449].log_data[15].valid := 1, [449].log_data[16].valid := 1, [449].log_data[17].valid := 1, [449].log_data[18].valid := 1, [449].log_data[19].valid := 1, [449].time.Year := 2023, [449].time.Month := 1, [449].time.Day := 12, [449].time.Hour := 8, [449].time.Minute := 44, [449].time.Second := 59, [450].log_data[0].min := 1.0, [450].log_data[0].max := 1.0, [450].log_data[0].total := 900.0, [450].log_data[0].time := 900.0, [450].log_data[0].minminute := 45, [450].log_data[0].maxminute := 45, [450].log_data[0].valid := 1, [450].log_data[1].valid := 1, [450].log_data[2].valid := 1,
        [450].log_data[3].valid := 1, [450].log_data[4].valid := 1, [450].log_data[5].valid := 1, [450].log_data[6].valid := 1, [450].log_data[7].valid := 1, [450].log_data[8].valid := 1, [450].log_data[9].valid := 1, [450].log_data[10].valid := 1, [450].log_data[11].valid := 1, [450].log_data[12].valid := 1, [450].log_data[13].valid := 1, [450].log_data[14].valid := 1, [450].log_data[15].valid := 1, [450].log_data[16].valid := 1, [450].log_data[17].valid := 1, [450].log_data[18].valid := 1, [450].log_data[19].valid := 1, [450].time.Year := 2023, [450].time.Month := 1, [450].time.Day := 12, [450].time.Hour := 8, [450].time.Minute := 59, [450].time.Second := 59, [451].log_data[0].min := 1.0, [451].log_data[0].max := 1.0, [451].log_data[0].total := 900.0, [451].log_data[0].time := 900.0, [451].log_data[0].valid := 1, [451].log_data[1].valid := 1, [451].log_data[2].valid := 1, [451].log_data[3].valid := 1, [451].log_data[4].valid := 1, [451].log_data[5].valid := 1, [451].log_data[6].valid := 1, [451].log_data[7].valid := 1, [451].log_data[8].valid := 1, [451].log_data[9].valid := 1, [451].log_data[10].valid := 1, [451].log_data[11].valid := 1, [451].log_data[12].valid := 1, [451].log_data[13].valid := 1, [451].log_data[14].valid := 1, [451].log_data[15].valid := 1, [451].log_data[16].valid := 1, [451].log_data[17].valid := 1, [451].log_data[18].valid := 1, [451].log_data[19].valid := 1, [451].time.Year := 2023, [451].time.Month := 1, [451].time.Day := 12, [451].time.Hour := 9, [451].time.Minute := 14, [451].time.Second := 59, [452].log_data[0].min := 1.0, [452].log_data[0].max := 1.0, [452].log_data[0].total := 900.0, [452].log_data[0].time := 900.0, [452].log_data[0].minminute := 15, [452].log_data[0].maxminute := 15, [452].log_data[0].valid := 1,
        [452].log_data[1].valid := 1, [452].log_data[2].valid := 1, [452].log_data[3].valid := 1, [452].log_data[4].valid := 1, [452].log_data[5].valid := 1, [452].log_data[6].valid := 1, [452].log_data[7].valid := 1, [452].log_data[8].valid := 1, [452].log_data[9].valid := 1, [452].log_data[10].valid := 1, [452].log_data[11].valid := 1, [452].log_data[12].valid := 1, [452].log_data[13].valid := 1, [452].log_data[14].valid := 1, [452].log_data[15].valid := 1, [452].log_data[16].valid := 1, [452].log_data[17].valid := 1, [452].log_data[18].valid := 1, [452].log_data[19].valid := 1, [452].time.Year := 2023, [452].time.Month := 1, [452].time.Day := 12, [452].time.Hour := 9, [452].time.Minute := 29, [452].time.Second := 59, [453].log_data[0].min := 1.0, [453].log_data[0].max := 1.0, [453].log_data[0].total := 900.0, [453].log_data[0].time := 900.0, [453].log_data[0].minminute := 30, [453].log_data[0].maxminute := 30, [453].log_data[0].valid := 1, [453].log_data[1].valid := 1, [453].log_data[2].valid := 1, [453].log_data[3].valid := 1, [453].log_data[4].valid := 1, [453].log_data[5].valid := 1, [453].log_data[6].valid := 1, [453].log_data[7].valid := 1, [453].log_data[8].valid := 1, [453].log_data[9].valid := 1, [453].log_data[10].valid := 1, [453].log_data[11].valid := 1, [453].log_data[12].valid := 1, [453].log_data[13].valid := 1, [453].log_data[14].valid := 1, [453].log_data[15].valid := 1, [453].log_data[16].valid := 1, [453].log_data[17].valid := 1, [453].log_data[18].valid := 1, [453].log_data[19].valid := 1, [453].time.Year := 2023, [453].time.Month := 1, [453].time.Day := 12, [453].time.Hour := 9, [453].time.Minute := 44, [453].time.Second := 59, [454].log_data[0].min := 1.0, [454].log_data[0].max := 1.0, [454].log_data[0].total := 900.0,
        [454].log_data[0].time := 900.0, [454].log_data[0].minminute := 45, [454].log_data[0].maxminute := 45, [454].log_data[0].valid := 1, [454].log_data[1].valid := 1, [454].log_data[2].valid := 1, [454].log_data[3].valid := 1, [454].log_data[4].valid := 1, [454].log_data[5].valid := 1, [454].log_data[6].valid := 1, [454].log_data[7].valid := 1, [454].log_data[8].valid := 1, [454].log_data[9].valid := 1, [454].log_data[10].valid := 1, [454].log_data[11].valid := 1, [454].log_data[12].valid := 1, [454].log_data[13].valid := 1, [454].log_data[14].valid := 1, [454].log_data[15].valid := 1, [454].log_data[16].valid := 1, [454].log_data[17].valid := 1, [454].log_data[18].valid := 1, [454].log_data[19].valid := 1, [454].time.Year := 2023, [454].time.Month := 1, [454].time.Day := 12, [454].time.Hour := 9, [454].time.Minute := 59, [454].time.Second := 59, [455].log_data[0].min := 1.0, [455].log_data[0].max := 1.0, [455].log_data[0].total := 900.0, [455].log_data[0].time := 900.0, [455].log_data[0].valid := 1, [455].log_data[1].valid := 1, [455].log_data[2].valid := 1, [455].log_data[3].valid := 1, [455].log_data[4].valid := 1, [455].log_data[5].valid := 1, [455].log_data[6].valid := 1, [455].log_data[7].valid := 1, [455].log_data[8].valid := 1, [455].log_data[9].valid := 1, [455].log_data[10].valid := 1, [455].log_data[11].valid := 1, [455].log_data[12].valid := 1, [455].log_data[13].valid := 1, [455].log_data[14].valid := 1, [455].log_data[15].valid := 1, [455].log_data[16].valid := 1, [455].log_data[17].valid := 1, [455].log_data[18].valid := 1, [455].log_data[19].valid := 1, [455].time.Year := 2023, [455].time.Month := 1, [455].time.Day := 12, [455].time.Hour := 10, [455].time.Minute := 14, [455].time.Second := 59, [456].log_data[0].min := 1.0,
        [456].log_data[0].max := 1.0, [456].log_data[0].total := 900.0, [456].log_data[0].time := 900.0, [456].log_data[0].minminute := 15, [456].log_data[0].maxminute := 15, [456].log_data[0].valid := 1, [456].log_data[1].valid := 1, [456].log_data[2].valid := 1, [456].log_data[3].valid := 1, [456].log_data[4].valid := 1, [456].log_data[5].valid := 1, [456].log_data[6].valid := 1, [456].log_data[7].valid := 1, [456].log_data[8].valid := 1, [456].log_data[9].valid := 1, [456].log_data[10].valid := 1, [456].log_data[11].valid := 1, [456].log_data[12].valid := 1, [456].log_data[13].valid := 1, [456].log_data[14].valid := 1, [456].log_data[15].valid := 1, [456].log_data[16].valid := 1, [456].log_data[17].valid := 1, [456].log_data[18].valid := 1, [456].log_data[19].valid := 1, [456].time.Year := 2023, [456].time.Month := 1, [456].time.Day := 12, [456].time.Hour := 10, [456].time.Minute := 29, [456].time.Second := 59, [457].log_data[0].min := 1.0, [457].log_data[0].max := 1.0, [457].log_data[0].total := 900.0, [457].log_data[0].time := 900.0, [457].log_data[0].minminute := 30, [457].log_data[0].maxminute := 30, [457].log_data[0].valid := 1, [457].log_data[1].valid := 1, [457].log_data[2].valid := 1, [457].log_data[3].valid := 1, [457].log_data[4].valid := 1, [457].log_data[5].valid := 1, [457].log_data[6].valid := 1, [457].log_data[7].valid := 1, [457].log_data[8].valid := 1, [457].log_data[9].valid := 1, [457].log_data[10].valid := 1, [457].log_data[11].valid := 1, [457].log_data[12].valid := 1, [457].log_data[13].valid := 1, [457].log_data[14].valid := 1, [457].log_data[15].valid := 1, [457].log_data[16].valid := 1, [457].log_data[17].valid := 1, [457].log_data[18].valid := 1, [457].log_data[19].valid := 1, [457].time.Year := 2023, [457].time.Month := 1, [457].time.Day := 12,
        [457].time.Hour := 10, [457].time.Minute := 44, [457].time.Second := 59, [458].log_data[0].min := 1.0, [458].log_data[0].max := 1.0, [458].log_data[0].total := 900.0, [458].log_data[0].time := 900.0, [458].log_data[0].minminute := 45, [458].log_data[0].maxminute := 45, [458].log_data[0].valid := 1, [458].log_data[1].valid := 1, [458].log_data[2].valid := 1, [458].log_data[3].valid := 1, [458].log_data[4].valid := 1, [458].log_data[5].valid := 1, [458].log_data[6].valid := 1, [458].log_data[7].valid := 1, [458].log_data[8].valid := 1, [458].log_data[9].valid := 1, [458].log_data[10].valid := 1, [458].log_data[11].valid := 1, [458].log_data[12].valid := 1, [458].log_data[13].valid := 1, [458].log_data[14].valid := 1, [458].log_data[15].valid := 1, [458].log_data[16].valid := 1, [458].log_data[17].valid := 1, [458].log_data[18].valid := 1, [458].log_data[19].valid := 1, [458].time.Year := 2023, [458].time.Month := 1, [458].time.Day := 12, [458].time.Hour := 10, [458].time.Minute := 59, [458].time.Second := 59, [459].log_data[0].min := 1.0, [459].log_data[0].max := 1.0, [459].log_data[0].total := 900.0, [459].log_data[0].time := 900.0, [459].log_data[0].valid := 1, [459].log_data[1].valid := 1, [459].log_data[2].valid := 1, [459].log_data[3].valid := 1, [459].log_data[4].valid := 1, [459].log_data[5].valid := 1, [459].log_data[6].valid := 1, [459].log_data[7].valid := 1, [459].log_data[8].valid := 1, [459].log_data[9].valid := 1, [459].log_data[10].valid := 1, [459].log_data[11].valid := 1, [459].log_data[12].valid := 1, [459].log_data[13].valid := 1, [459].log_data[14].valid := 1, [459].log_data[15].valid := 1, [459].log_data[16].valid := 1, [459].log_data[17].valid := 1, [459].log_data[18].valid := 1, [459].log_data[19].valid := 1, [459].time.Year := 2023,
        [459].time.Month := 1, [459].time.Day := 12, [459].time.Hour := 11, [459].time.Minute := 14, [459].time.Second := 59, [460].log_data[0].min := 1.0, [460].log_data[0].max := 1.0, [460].log_data[0].total := 900.0, [460].log_data[0].time := 900.0, [460].log_data[0].minminute := 15, [460].log_data[0].maxminute := 15, [460].log_data[0].valid := 1, [460].log_data[1].valid := 1, [460].log_data[2].valid := 1, [460].log_data[3].valid := 1, [460].log_data[4].valid := 1, [460].log_data[5].valid := 1, [460].log_data[6].valid := 1, [460].log_data[7].valid := 1, [460].log_data[8].valid := 1, [460].log_data[9].valid := 1, [460].log_data[10].valid := 1, [460].log_data[11].valid := 1, [460].log_data[12].valid := 1, [460].log_data[13].valid := 1, [460].log_data[14].valid := 1, [460].log_data[15].valid := 1, [460].log_data[16].valid := 1, [460].log_data[17].valid := 1, [460].log_data[18].valid := 1, [460].log_data[19].valid := 1, [460].time.Year := 2023, [460].time.Month := 1, [460].time.Day := 12, [460].time.Hour := 11, [460].time.Minute := 29, [460].time.Second := 59, [461].log_data[0].min := 1.0, [461].log_data[0].max := 1.0, [461].log_data[0].total := 900.0, [461].log_data[0].time := 900.0, [461].log_data[0].minminute := 30, [461].log_data[0].maxminute := 30, [461].log_data[0].valid := 1, [461].log_data[1].valid := 1, [461].log_data[2].valid := 1, [461].log_data[3].valid := 1, [461].log_data[4].valid := 1, [461].log_data[5].valid := 1, [461].log_data[6].valid := 1, [461].log_data[7].valid := 1, [461].log_data[8].valid := 1, [461].log_data[9].valid := 1, [461].log_data[10].valid := 1, [461].log_data[11].valid := 1, [461].log_data[12].valid := 1, [461].log_data[13].valid := 1, [461].log_data[14].valid := 1, [461].log_data[15].valid := 1, [461].log_data[16].valid := 1,
        [461].log_data[17].valid := 1, [461].log_data[18].valid := 1, [461].log_data[19].valid := 1, [461].time.Year := 2023, [461].time.Month := 1, [461].time.Day := 12, [461].time.Hour := 11, [461].time.Minute := 44, [461].time.Second := 59, [462].log_data[0].min := 1.0, [462].log_data[0].max := 1.0, [462].log_data[0].total := 900.0, [462].log_data[0].time := 900.0, [462].log_data[0].minminute := 45, [462].log_data[0].maxminute := 45, [462].log_data[0].valid := 1, [462].log_data[1].valid := 1, [462].log_data[2].valid := 1, [462].log_data[3].valid := 1, [462].log_data[4].valid := 1, [462].log_data[5].valid := 1, [462].log_data[6].valid := 1, [462].log_data[7].valid := 1, [462].log_data[8].valid := 1, [462].log_data[9].valid := 1, [462].log_data[10].valid := 1, [462].log_data[11].valid := 1, [462].log_data[12].valid := 1, [462].log_data[13].valid := 1, [462].log_data[14].valid := 1, [462].log_data[15].valid := 1, [462].log_data[16].valid := 1, [462].log_data[17].valid := 1, [462].log_data[18].valid := 1, [462].log_data[19].valid := 1, [462].time.Year := 2023, [462].time.Month := 1, [462].time.Day := 12, [462].time.Hour := 11, [462].time.Minute := 59, [462].time.Second := 59, [463].log_data[0].min := 1.0, [463].log_data[0].max := 1.0, [463].log_data[0].total := 900.0, [463].log_data[0].time := 900.0, [463].log_data[0].valid := 1, [463].log_data[1].valid := 1, [463].log_data[2].valid := 1, [463].log_data[3].valid := 1, [463].log_data[4].valid := 1, [463].log_data[5].valid := 1, [463].log_data[6].valid := 1, [463].log_data[7].valid := 1, [463].log_data[8].valid := 1, [463].log_data[9].valid := 1, [463].log_data[10].valid := 1, [463].log_data[11].valid := 1, [463].log_data[12].valid := 1, [463].log_data[13].valid := 1, [463].log_data[14].valid := 1,
        [463].log_data[15].valid := 1, [463].log_data[16].valid := 1, [463].log_data[17].valid := 1, [463].log_data[18].valid := 1, [463].log_data[19].valid := 1, [463].time.Year := 2023, [463].time.Month := 1, [463].time.Day := 12, [463].time.Hour := 12, [463].time.Minute := 14, [463].time.Second := 59, [464].log_data[0].min := 1.0, [464].log_data[0].max := 1.0, [464].log_data[0].total := 900.0, [464].log_data[0].time := 900.0, [464].log_data[0].minminute := 15, [464].log_data[0].maxminute := 15, [464].log_data[0].valid := 1, [464].log_data[1].valid := 1, [464].log_data[2].valid := 1, [464].log_data[3].valid := 1, [464].log_data[4].valid := 1, [464].log_data[5].valid := 1, [464].log_data[6].valid := 1, [464].log_data[7].valid := 1, [464].log_data[8].valid := 1, [464].log_data[9].valid := 1, [464].log_data[10].valid := 1, [464].log_data[11].valid := 1, [464].log_data[12].valid := 1, [464].log_data[13].valid := 1, [464].log_data[14].valid := 1, [464].log_data[15].valid := 1, [464].log_data[16].valid := 1, [464].log_data[17].valid := 1, [464].log_data[18].valid := 1, [464].log_data[19].valid := 1, [464].time.Year := 2023, [464].time.Month := 1, [464].time.Day := 12, [464].time.Hour := 12, [464].time.Minute := 29, [464].time.Second := 59, [465].log_data[0].min := 1.0, [465].log_data[0].max := 1.0, [465].log_data[0].total := 900.0, [465].log_data[0].time := 900.0, [465].log_data[0].minminute := 30, [465].log_data[0].maxminute := 30, [465].log_data[0].valid := 1, [465].log_data[1].valid := 1, [465].log_data[2].valid := 1, [465].log_data[3].valid := 1, [465].log_data[4].valid := 1, [465].log_data[5].valid := 1, [465].log_data[6].valid := 1, [465].log_data[7].valid := 1, [465].log_data[8].valid := 1, [465].log_data[9].valid := 1, [465].log_data[10].valid := 1,
        [465].log_data[11].valid := 1, [465].log_data[12].valid := 1, [465].log_data[13].valid := 1, [465].log_data[14].valid := 1, [465].log_data[15].valid := 1, [465].log_data[16].valid := 1, [465].log_data[17].valid := 1, [465].log_data[18].valid := 1, [465].log_data[19].valid := 1, [465].time.Year := 2023, [465].time.Month := 1, [465].time.Day := 12, [465].time.Hour := 12, [465].time.Minute := 44, [465].time.Second := 59, [466].log_data[0].min := 1.0, [466].log_data[0].max := 1.0, [466].log_data[0].total := 900.0, [466].log_data[0].time := 900.0, [466].log_data[0].minminute := 45, [466].log_data[0].maxminute := 45, [466].log_data[0].valid := 1, [466].log_data[1].valid := 1, [466].log_data[2].valid := 1, [466].log_data[3].valid := 1, [466].log_data[4].valid := 1, [466].log_data[5].valid := 1, [466].log_data[6].valid := 1, [466].log_data[7].valid := 1, [466].log_data[8].valid := 1, [466].log_data[9].valid := 1, [466].log_data[10].valid := 1, [466].log_data[11].valid := 1, [466].log_data[12].valid := 1, [466].log_data[13].valid := 1, [466].log_data[14].valid := 1, [466].log_data[15].valid := 1, [466].log_data[16].valid := 1, [466].log_data[17].valid := 1, [466].log_data[18].valid := 1, [466].log_data[19].valid := 1, [466].time.Year := 2023, [466].time.Month := 1, [466].time.Day := 12, [466].time.Hour := 12, [466].time.Minute := 59, [466].time.Second := 59, [467].log_data[0].min := 1.0, [467].log_data[0].max := 1.0, [467].log_data[0].total := 899.5, [467].log_data[0].time := 899.5, [467].log_data[0].valid := 1, [467].log_data[1].valid := 1, [467].log_data[2].valid := 1, [467].log_data[3].valid := 1, [467].log_data[4].valid := 1, [467].log_data[5].valid := 1, [467].log_data[6].valid := 1, [467].log_data[7].valid := 1, [467].log_data[8].valid := 1,
        [467].log_data[9].valid := 1, [467].log_data[10].valid := 1, [467].log_data[11].valid := 1, [467].log_data[12].valid := 1, [467].log_data[13].valid := 1, [467].log_data[14].valid := 1, [467].log_data[15].valid := 1, [467].log_data[16].valid := 1, [467].log_data[17].valid := 1, [467].log_data[18].valid := 1, [467].log_data[19].valid := 1, [467].time.Year := 2023, [467].time.Month := 1, [467].time.Day := 12, [467].time.Hour := 13, [467].time.Minute := 14, [467].time.Second := 59, [468].log_data[0].min := 1.0, [468].log_data[0].max := 1.0, [468].log_data[0].total := 900.0, [468].log_data[0].time := 900.0, [468].log_data[0].minminute := 15, [468].log_data[0].maxminute := 15, [468].log_data[0].valid := 1, [468].log_data[1].valid := 1, [468].log_data[2].valid := 1, [468].log_data[3].valid := 1, [468].log_data[4].valid := 1, [468].log_data[5].valid := 1, [468].log_data[6].valid := 1, [468].log_data[7].valid := 1, [468].log_data[8].valid := 1, [468].log_data[9].valid := 1, [468].log_data[10].valid := 1, [468].log_data[11].valid := 1, [468].log_data[12].valid := 1, [468].log_data[13].valid := 1, [468].log_data[14].valid := 1, [468].log_data[15].valid := 1, [468].log_data[16].valid := 1, [468].log_data[17].valid := 1, [468].log_data[18].valid := 1, [468].log_data[19].valid := 1, [468].time.Year := 2023, [468].time.Month := 1, [468].time.Day := 12, [468].time.Hour := 13, [468].time.Minute := 29, [468].time.Second := 59, [469].log_data[0].min := 1.0, [469].log_data[0].max := 1.0, [469].log_data[0].total := 900.0, [469].log_data[0].time := 900.0, [469].log_data[0].minminute := 30, [469].log_data[0].maxminute := 30, [469].log_data[0].valid := 1, [469].log_data[1].valid := 1, [469].log_data[2].valid := 1, [469].log_data[3].valid := 1, [469].log_data[4].valid := 1,
        [469].log_data[5].valid := 1, [469].log_data[6].valid := 1, [469].log_data[7].valid := 1, [469].log_data[8].valid := 1, [469].log_data[9].valid := 1, [469].log_data[10].valid := 1, [469].log_data[11].valid := 1, [469].log_data[12].valid := 1, [469].log_data[13].valid := 1, [469].log_data[14].valid := 1, [469].log_data[15].valid := 1, [469].log_data[16].valid := 1, [469].log_data[17].valid := 1, [469].log_data[18].valid := 1, [469].log_data[19].valid := 1, [469].time.Year := 2023, [469].time.Month := 1, [469].time.Day := 12, [469].time.Hour := 13, [469].time.Minute := 44, [469].time.Second := 59, [470].log_data[0].min := 1.0, [470].log_data[0].max := 1.0, [470].log_data[0].total := 900.0, [470].log_data[0].time := 900.0, [470].log_data[0].minminute := 45, [470].log_data[0].maxminute := 45, [470].log_data[0].valid := 1, [470].log_data[1].valid := 1, [470].log_data[2].valid := 1, [470].log_data[3].valid := 1, [470].log_data[4].valid := 1, [470].log_data[5].valid := 1, [470].log_data[6].valid := 1, [470].log_data[7].valid := 1, [470].log_data[8].valid := 1, [470].log_data[9].valid := 1, [470].log_data[10].valid := 1, [470].log_data[11].valid := 1, [470].log_data[12].valid := 1, [470].log_data[13].valid := 1, [470].log_data[14].valid := 1, [470].log_data[15].valid := 1, [470].log_data[16].valid := 1, [470].log_data[17].valid := 1, [470].log_data[18].valid := 1, [470].log_data[19].valid := 1, [470].time.Year := 2023, [470].time.Month := 1, [470].time.Day := 12, [470].time.Hour := 13, [470].time.Minute := 59, [470].time.Second := 59, [471].log_data[0].min := 1.0, [471].log_data[0].max := 1.0, [471].log_data[0].total := 900.0, [471].log_data[0].time := 900.0, [471].log_data[0].valid := 1, [471].log_data[1].valid := 1, [471].log_data[2].valid := 1,
        [471].log_data[3].valid := 1, [471].log_data[4].valid := 1, [471].log_data[5].valid := 1, [471].log_data[6].valid := 1, [471].log_data[7].valid := 1, [471].log_data[8].valid := 1, [471].log_data[9].valid := 1, [471].log_data[10].valid := 1, [471].log_data[11].valid := 1, [471].log_data[12].valid := 1, [471].log_data[13].valid := 1, [471].log_data[14].valid := 1, [471].log_data[15].valid := 1, [471].log_data[16].valid := 1, [471].log_data[17].valid := 1, [471].log_data[18].valid := 1, [471].log_data[19].valid := 1, [471].time.Year := 2023, [471].time.Month := 1, [471].time.Day := 12, [471].time.Hour := 14, [471].time.Minute := 14, [471].time.Second := 59, [472].log_data[0].min := 1.0, [472].log_data[0].max := 1.0, [472].log_data[0].total := 900.0, [472].log_data[0].time := 900.0, [472].log_data[0].minminute := 15, [472].log_data[0].maxminute := 15, [472].log_data[0].valid := 1, [472].log_data[1].valid := 1, [472].log_data[2].valid := 1, [472].log_data[3].valid := 1, [472].log_data[4].valid := 1, [472].log_data[5].valid := 1, [472].log_data[6].valid := 1, [472].log_data[7].valid := 1, [472].log_data[8].valid := 1, [472].log_data[9].valid := 1, [472].log_data[10].valid := 1, [472].log_data[11].valid := 1, [472].log_data[12].valid := 1, [472].log_data[13].valid := 1, [472].log_data[14].valid := 1, [472].log_data[15].valid := 1, [472].log_data[16].valid := 1, [472].log_data[17].valid := 1, [472].log_data[18].valid := 1, [472].log_data[19].valid := 1, [472].time.Year := 2023, [472].time.Month := 1, [472].time.Day := 12, [472].time.Hour := 14, [472].time.Minute := 29, [472].time.Second := 59, [473].log_data[0].min := 1.0, [473].log_data[0].max := 1.0, [473].log_data[0].total := 900.0, [473].log_data[0].time := 900.0, [473].log_data[0].minminute := 30,
        [473].log_data[0].maxminute := 30, [473].log_data[0].valid := 1, [473].log_data[1].valid := 1, [473].log_data[2].valid := 1, [473].log_data[3].valid := 1, [473].log_data[4].valid := 1, [473].log_data[5].valid := 1, [473].log_data[6].valid := 1, [473].log_data[7].valid := 1, [473].log_data[8].valid := 1, [473].log_data[9].valid := 1, [473].log_data[10].valid := 1, [473].log_data[11].valid := 1, [473].log_data[12].valid := 1, [473].log_data[13].valid := 1, [473].log_data[14].valid := 1, [473].log_data[15].valid := 1, [473].log_data[16].valid := 1, [473].log_data[17].valid := 1, [473].log_data[18].valid := 1, [473].log_data[19].valid := 1, [473].time.Year := 2023, [473].time.Month := 1, [473].time.Day := 12, [473].time.Hour := 14, [473].time.Minute := 44, [473].time.Second := 59, [474].log_data[0].min := 1.0, [474].log_data[0].max := 1.0, [474].log_data[0].total := 900.0, [474].log_data[0].time := 900.0, [474].log_data[0].minminute := 45, [474].log_data[0].maxminute := 45, [474].log_data[0].valid := 1, [474].log_data[1].valid := 1, [474].log_data[2].valid := 1, [474].log_data[3].valid := 1, [474].log_data[4].valid := 1, [474].log_data[5].valid := 1, [474].log_data[6].valid := 1, [474].log_data[7].valid := 1, [474].log_data[8].valid := 1, [474].log_data[9].valid := 1, [474].log_data[10].valid := 1, [474].log_data[11].valid := 1, [474].log_data[12].valid := 1, [474].log_data[13].valid := 1, [474].log_data[14].valid := 1, [474].log_data[15].valid := 1, [474].log_data[16].valid := 1, [474].log_data[17].valid := 1, [474].log_data[18].valid := 1, [474].log_data[19].valid := 1, [474].time.Year := 2023, [474].time.Month := 1, [474].time.Day := 12, [474].time.Hour := 14, [474].time.Minute := 59, [474].time.Second := 59, [475].log_data[0].min := 1.0,
        [475].log_data[0].max := 1.0, [475].log_data[0].total := 900.0, [475].log_data[0].time := 900.0, [475].log_data[0].valid := 1, [475].log_data[1].valid := 1, [475].log_data[2].valid := 1, [475].log_data[3].valid := 1, [475].log_data[4].valid := 1, [475].log_data[5].valid := 1, [475].log_data[6].valid := 1, [475].log_data[7].valid := 1, [475].log_data[8].valid := 1, [475].log_data[9].valid := 1, [475].log_data[10].valid := 1, [475].log_data[11].valid := 1, [475].log_data[12].valid := 1, [475].log_data[13].valid := 1, [475].log_data[14].valid := 1, [475].log_data[15].valid := 1, [475].log_data[16].valid := 1, [475].log_data[17].valid := 1, [475].log_data[18].valid := 1, [475].log_data[19].valid := 1, [475].time.Year := 2023, [475].time.Month := 1, [475].time.Day := 12, [475].time.Hour := 15, [475].time.Minute := 14, [475].time.Second := 59, [476].log_data[0].min := 1.0, [476].log_data[0].max := 1.0, [476].log_data[0].total := 900.0, [476].log_data[0].time := 900.0, [476].log_data[0].minminute := 15, [476].log_data[0].maxminute := 15, [476].log_data[0].valid := 1, [476].log_data[1].valid := 1, [476].log_data[2].valid := 1, [476].log_data[3].valid := 1, [476].log_data[4].valid := 1, [476].log_data[5].valid := 1, [476].log_data[6].valid := 1, [476].log_data[7].valid := 1, [476].log_data[8].valid := 1, [476].log_data[9].valid := 1, [476].log_data[10].valid := 1, [476].log_data[11].valid := 1, [476].log_data[12].valid := 1, [476].log_data[13].valid := 1, [476].log_data[14].valid := 1, [476].log_data[15].valid := 1, [476].log_data[16].valid := 1, [476].log_data[17].valid := 1, [476].log_data[18].valid := 1, [476].log_data[19].valid := 1, [476].time.Year := 2023, [476].time.Month := 1, [476].time.Day := 12, [476].time.Hour := 15, [476].time.Minute := 29,
        [476].time.Second := 59, [477].log_data[0].min := 1.0, [477].log_data[0].max := 1.0, [477].log_data[0].total := 900.0, [477].log_data[0].time := 900.0, [477].log_data[0].minminute := 30, [477].log_data[0].maxminute := 30, [477].log_data[0].valid := 1, [477].log_data[1].valid := 1, [477].log_data[2].valid := 1, [477].log_data[3].valid := 1, [477].log_data[4].valid := 1, [477].log_data[5].valid := 1, [477].log_data[6].valid := 1, [477].log_data[7].valid := 1, [477].log_data[8].valid := 1, [477].log_data[9].valid := 1, [477].log_data[10].valid := 1, [477].log_data[11].valid := 1, [477].log_data[12].valid := 1, [477].log_data[13].valid := 1, [477].log_data[14].valid := 1, [477].log_data[15].valid := 1, [477].log_data[16].valid := 1, [477].log_data[17].valid := 1, [477].log_data[18].valid := 1, [477].log_data[19].valid := 1, [477].time.Year := 2023, [477].time.Month := 1, [477].time.Day := 12, [477].time.Hour := 15, [477].time.Minute := 44, [477].time.Second := 59, [478].log_data[0].min := 1.0, [478].log_data[0].max := 1.0, [478].log_data[0].total := 900.0, [478].log_data[0].time := 900.0, [478].log_data[0].minminute := 45, [478].log_data[0].maxminute := 45, [478].log_data[0].valid := 1, [478].log_data[1].valid := 1, [478].log_data[2].valid := 1, [478].log_data[3].valid := 1, [478].log_data[4].valid := 1, [478].log_data[5].valid := 1, [478].log_data[6].valid := 1, [478].log_data[7].valid := 1, [478].log_data[8].valid := 1, [478].log_data[9].valid := 1, [478].log_data[10].valid := 1, [478].log_data[11].valid := 1, [478].log_data[12].valid := 1, [478].log_data[13].valid := 1, [478].log_data[14].valid := 1, [478].log_data[15].valid := 1, [478].log_data[16].valid := 1, [478].log_data[17].valid := 1, [478].log_data[18].valid := 1, [478].log_data[19].valid := 1, [478].time.Year := 2023,
        [478].time.Month := 1, [478].time.Day := 12, [478].time.Hour := 15, [478].time.Minute := 59, [478].time.Second := 59, [479].log_data[0].min := 1.0, [479].log_data[0].max := 1.0, [479].log_data[0].total := 900.0, [479].log_data[0].time := 900.0, [479].log_data[0].valid := 1, [479].log_data[1].valid := 1, [479].log_data[2].valid := 1, [479].log_data[3].valid := 1, [479].log_data[4].valid := 1, [479].log_data[5].valid := 1, [479].log_data[6].valid := 1, [479].log_data[7].valid := 1, [479].log_data[8].valid := 1, [479].log_data[9].valid := 1, [479].log_data[10].valid := 1, [479].log_data[11].valid := 1, [479].log_data[12].valid := 1, [479].log_data[13].valid := 1, [479].log_data[14].valid := 1, [479].log_data[15].valid := 1, [479].log_data[16].valid := 1, [479].log_data[17].valid := 1, [479].log_data[18].valid := 1, [479].log_data[19].valid := 1, [479].time.Year := 2023, [479].time.Month := 1, [479].time.Day := 12, [479].time.Hour := 16, [479].time.Minute := 14, [479].time.Second := 59, [480].log_data[0].min := 1.0, [480].log_data[0].max := 1.0, [480].log_data[0].total := 900.0, [480].log_data[0].time := 900.0, [480].log_data[0].minminute := 15, [480].log_data[0].maxminute := 15, [480].log_data[0].valid := 1, [480].log_data[1].valid := 1, [480].log_data[2].valid := 1, [480].log_data[3].valid := 1, [480].log_data[4].valid := 1, [480].log_data[5].valid := 1, [480].log_data[6].valid := 1, [480].log_data[7].valid := 1, [480].log_data[8].valid := 1, [480].log_data[9].valid := 1, [480].log_data[10].valid := 1, [480].log_data[11].valid := 1, [480].log_data[12].valid := 1, [480].log_data[13].valid := 1, [480].log_data[14].valid := 1, [480].log_data[15].valid := 1, [480].log_data[16].valid := 1, [480].log_data[17].valid := 1, [480].log_data[18].valid := 1,
        [480].log_data[19].valid := 1, [480].time.Year := 2023, [480].time.Month := 1, [480].time.Day := 12, [480].time.Hour := 16, [480].time.Minute := 29, [480].time.Second := 59, [481].log_data[0].min := 1.0, [481].log_data[0].max := 1.0, [481].log_data[0].total := 900.0, [481].log_data[0].time := 900.0, [481].log_data[0].minminute := 30, [481].log_data[0].maxminute := 30, [481].log_data[0].valid := 1, [481].log_data[1].valid := 1, [481].log_data[2].valid := 1, [481].log_data[3].valid := 1, [481].log_data[4].valid := 1, [481].log_data[5].valid := 1, [481].log_data[6].valid := 1, [481].log_data[7].valid := 1, [481].log_data[8].valid := 1, [481].log_data[9].valid := 1, [481].log_data[10].valid := 1, [481].log_data[11].valid := 1, [481].log_data[12].valid := 1, [481].log_data[13].valid := 1, [481].log_data[14].valid := 1, [481].log_data[15].valid := 1, [481].log_data[16].valid := 1, [481].log_data[17].valid := 1, [481].log_data[18].valid := 1, [481].log_data[19].valid := 1, [481].time.Year := 2023, [481].time.Month := 1, [481].time.Day := 12, [481].time.Hour := 16, [481].time.Minute := 44, [481].time.Second := 59, [482].log_data[0].min := 1.0, [482].log_data[0].max := 1.0, [482].log_data[0].total := 900.0, [482].log_data[0].time := 900.0, [482].log_data[0].minminute := 45, [482].log_data[0].maxminute := 45, [482].log_data[0].valid := 1, [482].log_data[1].valid := 1, [482].log_data[2].valid := 1, [482].log_data[3].valid := 1, [482].log_data[4].valid := 1, [482].log_data[5].valid := 1, [482].log_data[6].valid := 1, [482].log_data[7].valid := 1, [482].log_data[8].valid := 1, [482].log_data[9].valid := 1, [482].log_data[10].valid := 1, [482].log_data[11].valid := 1, [482].log_data[12].valid := 1, [482].log_data[13].valid := 1, [482].log_data[14].valid := 1,
        [482].log_data[15].valid := 1, [482].log_data[16].valid := 1, [482].log_data[17].valid := 1, [482].log_data[18].valid := 1, [482].log_data[19].valid := 1, [482].time.Year := 2023, [482].time.Month := 1, [482].time.Day := 12, [482].time.Hour := 16, [482].time.Minute := 59, [482].time.Second := 59, [483].log_data[0].min := 1.0, [483].log_data[0].max := 1.0, [483].log_data[0].total := 900.0, [483].log_data[0].time := 900.0, [483].log_data[0].valid := 1, [483].log_data[1].valid := 1, [483].log_data[2].valid := 1, [483].log_data[3].valid := 1, [483].log_data[4].valid := 1, [483].log_data[5].valid := 1, [483].log_data[6].valid := 1, [483].log_data[7].valid := 1, [483].log_data[8].valid := 1, [483].log_data[9].valid := 1, [483].log_data[10].valid := 1, [483].log_data[11].valid := 1, [483].log_data[12].valid := 1, [483].log_data[13].valid := 1, [483].log_data[14].valid := 1, [483].log_data[15].valid := 1, [483].log_data[16].valid := 1, [483].log_data[17].valid := 1, [483].log_data[18].valid := 1, [483].log_data[19].valid := 1, [483].time.Year := 2023, [483].time.Month := 1, [483].time.Day := 12, [483].time.Hour := 17, [483].time.Minute := 14, [483].time.Second := 59, [484].log_data[0].min := 1.0, [484].log_data[0].max := 1.0, [484].log_data[0].total := 900.0, [484].log_data[0].time := 900.0, [484].log_data[0].minminute := 15, [484].log_data[0].maxminute := 15, [484].log_data[0].valid := 1, [484].log_data[1].valid := 1, [484].log_data[2].valid := 1, [484].log_data[3].valid := 1, [484].log_data[4].valid := 1, [484].log_data[5].valid := 1, [484].log_data[6].valid := 1, [484].log_data[7].valid := 1, [484].log_data[8].valid := 1, [484].log_data[9].valid := 1, [484].log_data[10].valid := 1, [484].log_data[11].valid := 1, [484].log_data[12].valid := 1,
        [484].log_data[13].valid := 1, [484].log_data[14].valid := 1, [484].log_data[15].valid := 1, [484].log_data[16].valid := 1, [484].log_data[17].valid := 1, [484].log_data[18].valid := 1, [484].log_data[19].valid := 1, [484].time.Year := 2023, [484].time.Month := 1, [484].time.Day := 12, [484].time.Hour := 17, [484].time.Minute := 29, [484].time.Second := 59, [485].log_data[0].min := 1.0, [485].log_data[0].max := 1.0, [485].log_data[0].total := 900.0, [485].log_data[0].time := 900.0, [485].log_data[0].minminute := 30, [485].log_data[0].maxminute := 30, [485].log_data[0].valid := 1, [485].log_data[1].valid := 1, [485].log_data[2].valid := 1, [485].log_data[3].valid := 1, [485].log_data[4].valid := 1, [485].log_data[5].valid := 1, [485].log_data[6].valid := 1, [485].log_data[7].valid := 1, [485].log_data[8].valid := 1, [485].log_data[9].valid := 1, [485].log_data[10].valid := 1, [485].log_data[11].valid := 1, [485].log_data[12].valid := 1, [485].log_data[13].valid := 1, [485].log_data[14].valid := 1, [485].log_data[15].valid := 1, [485].log_data[16].valid := 1, [485].log_data[17].valid := 1, [485].log_data[18].valid := 1, [485].log_data[19].valid := 1, [485].time.Year := 2023, [485].time.Month := 1, [485].time.Day := 12, [485].time.Hour := 17, [485].time.Minute := 44, [485].time.Second := 59, [486].log_data[0].min := 1.0, [486].log_data[0].max := 1.0, [486].log_data[0].total := 900.0, [486].log_data[0].time := 900.0, [486].log_data[0].minminute := 45, [486].log_data[0].maxminute := 45, [486].log_data[0].valid := 1, [486].log_data[1].valid := 1, [486].log_data[2].valid := 1, [486].log_data[3].valid := 1, [486].log_data[4].valid := 1, [486].log_data[5].valid := 1, [486].log_data[6].valid := 1, [486].log_data[7].valid := 1, [486].log_data[8].valid := 1,
        [486].log_data[9].valid := 1, [486].log_data[10].valid := 1, [486].log_data[11].valid := 1, [486].log_data[12].valid := 1, [486].log_data[13].valid := 1, [486].log_data[14].valid := 1, [486].log_data[15].valid := 1, [486].log_data[16].valid := 1, [486].log_data[17].valid := 1, [486].log_data[18].valid := 1, [486].log_data[19].valid := 1, [486].time.Year := 2023, [486].time.Month := 1, [486].time.Day := 12, [486].time.Hour := 17, [486].time.Minute := 59, [486].time.Second := 59, [487].log_data[0].min := 1.0, [487].log_data[0].max := 1.0, [487].log_data[0].total := 900.0, [487].log_data[0].time := 900.0, [487].log_data[0].valid := 1, [487].log_data[1].valid := 1, [487].log_data[2].valid := 1, [487].log_data[3].valid := 1, [487].log_data[4].valid := 1, [487].log_data[5].valid := 1, [487].log_data[6].valid := 1, [487].log_data[7].valid := 1, [487].log_data[8].valid := 1, [487].log_data[9].valid := 1, [487].log_data[10].valid := 1, [487].log_data[11].valid := 1, [487].log_data[12].valid := 1, [487].log_data[13].valid := 1, [487].log_data[14].valid := 1, [487].log_data[15].valid := 1, [487].log_data[16].valid := 1, [487].log_data[17].valid := 1, [487].log_data[18].valid := 1, [487].log_data[19].valid := 1, [487].time.Year := 2023, [487].time.Month := 1, [487].time.Day := 12, [487].time.Hour := 18, [487].time.Minute := 14, [487].time.Second := 59, [488].log_data[0].min := 1.0, [488].log_data[0].max := 1.0, [488].log_data[0].total := 900.0, [488].log_data[0].time := 900.0, [488].log_data[0].minminute := 15, [488].log_data[0].maxminute := 15, [488].log_data[0].valid := 1, [488].log_data[1].valid := 1, [488].log_data[2].valid := 1, [488].log_data[3].valid := 1, [488].log_data[4].valid := 1, [488].log_data[5].valid := 1, [488].log_data[6].valid := 1,
        [488].log_data[7].valid := 1, [488].log_data[8].valid := 1, [488].log_data[9].valid := 1, [488].log_data[10].valid := 1, [488].log_data[11].valid := 1, [488].log_data[12].valid := 1, [488].log_data[13].valid := 1, [488].log_data[14].valid := 1, [488].log_data[15].valid := 1, [488].log_data[16].valid := 1, [488].log_data[17].valid := 1, [488].log_data[18].valid := 1, [488].log_data[19].valid := 1, [488].time.Year := 2023, [488].time.Month := 1, [488].time.Day := 12, [488].time.Hour := 18, [488].time.Minute := 29, [488].time.Second := 59, [489].log_data[0].min := 1.0, [489].log_data[0].max := 1.0, [489].log_data[0].total := 900.0, [489].log_data[0].time := 900.0, [489].log_data[0].minminute := 30, [489].log_data[0].maxminute := 30, [489].log_data[0].valid := 1, [489].log_data[1].valid := 1, [489].log_data[2].valid := 1, [489].log_data[3].valid := 1, [489].log_data[4].valid := 1, [489].log_data[5].valid := 1, [489].log_data[6].valid := 1, [489].log_data[7].valid := 1, [489].log_data[8].valid := 1, [489].log_data[9].valid := 1, [489].log_data[10].valid := 1, [489].log_data[11].valid := 1, [489].log_data[12].valid := 1, [489].log_data[13].valid := 1, [489].log_data[14].valid := 1, [489].log_data[15].valid := 1, [489].log_data[16].valid := 1, [489].log_data[17].valid := 1, [489].log_data[18].valid := 1, [489].log_data[19].valid := 1, [489].time.Year := 2023, [489].time.Month := 1, [489].time.Day := 12, [489].time.Hour := 18, [489].time.Minute := 44, [489].time.Second := 59, [490].log_data[0].min := 1.0, [490].log_data[0].max := 1.0, [490].log_data[0].total := 900.0, [490].log_data[0].time := 900.0, [490].log_data[0].minminute := 45, [490].log_data[0].maxminute := 45, [490].log_data[0].valid := 1, [490].log_data[1].valid := 1, [490].log_data[2].valid := 1,
        [490].log_data[3].valid := 1, [490].log_data[4].valid := 1, [490].log_data[5].valid := 1, [490].log_data[6].valid := 1, [490].log_data[7].valid := 1, [490].log_data[8].valid := 1, [490].log_data[9].valid := 1, [490].log_data[10].valid := 1, [490].log_data[11].valid := 1, [490].log_data[12].valid := 1, [490].log_data[13].valid := 1, [490].log_data[14].valid := 1, [490].log_data[15].valid := 1, [490].log_data[16].valid := 1, [490].log_data[17].valid := 1, [490].log_data[18].valid := 1, [490].log_data[19].valid := 1, [490].time.Year := 2023, [490].time.Month := 1, [490].time.Day := 12, [490].time.Hour := 18, [490].time.Minute := 59, [490].time.Second := 59, [491].log_data[0].min := 1.0, [491].log_data[0].max := 1.0, [491].log_data[0].total := 900.0, [491].log_data[0].time := 900.0, [491].log_data[0].valid := 1, [491].log_data[1].valid := 1, [491].log_data[2].valid := 1, [491].log_data[3].valid := 1, [491].log_data[4].valid := 1, [491].log_data[5].valid := 1, [491].log_data[6].valid := 1, [491].log_data[7].valid := 1, [491].log_data[8].valid := 1, [491].log_data[9].valid := 1, [491].log_data[10].valid := 1, [491].log_data[11].valid := 1, [491].log_data[12].valid := 1, [491].log_data[13].valid := 1, [491].log_data[14].valid := 1, [491].log_data[15].valid := 1, [491].log_data[16].valid := 1, [491].log_data[17].valid := 1, [491].log_data[18].valid := 1, [491].log_data[19].valid := 1, [491].time.Year := 2023, [491].time.Month := 1, [491].time.Day := 12, [491].time.Hour := 19, [491].time.Minute := 14, [491].time.Second := 59, [492].log_data[0].min := 1.0, [492].log_data[0].max := 1.0, [492].log_data[0].total := 900.0, [492].log_data[0].time := 900.0, [492].log_data[0].minminute := 15, [492].log_data[0].maxminute := 15, [492].log_data[0].valid := 1,
        [492].log_data[1].valid := 1, [492].log_data[2].valid := 1, [492].log_data[3].valid := 1, [492].log_data[4].valid := 1, [492].log_data[5].valid := 1, [492].log_data[6].valid := 1, [492].log_data[7].valid := 1, [492].log_data[8].valid := 1, [492].log_data[9].valid := 1, [492].log_data[10].valid := 1, [492].log_data[11].valid := 1, [492].log_data[12].valid := 1, [492].log_data[13].valid := 1, [492].log_data[14].valid := 1, [492].log_data[15].valid := 1, [492].log_data[16].valid := 1, [492].log_data[17].valid := 1, [492].log_data[18].valid := 1, [492].log_data[19].valid := 1, [492].time.Year := 2023, [492].time.Month := 1, [492].time.Day := 12, [492].time.Hour := 19, [492].time.Minute := 29, [492].time.Second := 59, [493].log_data[0].min := 1.0, [493].log_data[0].max := 1.0, [493].log_data[0].total := 900.0, [493].log_data[0].time := 900.0, [493].log_data[0].minminute := 30, [493].log_data[0].maxminute := 30, [493].log_data[0].valid := 1, [493].log_data[1].valid := 1, [493].log_data[2].valid := 1, [493].log_data[3].valid := 1, [493].log_data[4].valid := 1, [493].log_data[5].valid := 1, [493].log_data[6].valid := 1, [493].log_data[7].valid := 1, [493].log_data[8].valid := 1, [493].log_data[9].valid := 1, [493].log_data[10].valid := 1, [493].log_data[11].valid := 1, [493].log_data[12].valid := 1, [493].log_data[13].valid := 1, [493].log_data[14].valid := 1, [493].log_data[15].valid := 1, [493].log_data[16].valid := 1, [493].log_data[17].valid := 1, [493].log_data[18].valid := 1, [493].log_data[19].valid := 1, [493].time.Year := 2023, [493].time.Month := 1, [493].time.Day := 12, [493].time.Hour := 19, [493].time.Minute := 44, [493].time.Second := 59, [494].log_data[0].min := 1.0, [494].log_data[0].max := 1.0, [494].log_data[0].total := 900.0,
        [494].log_data[0].time := 900.0, [494].log_data[0].minminute := 45, [494].log_data[0].maxminute := 45, [494].log_data[0].valid := 1, [494].log_data[1].valid := 1, [494].log_data[2].valid := 1, [494].log_data[3].valid := 1, [494].log_data[4].valid := 1, [494].log_data[5].valid := 1, [494].log_data[6].valid := 1, [494].log_data[7].valid := 1, [494].log_data[8].valid := 1, [494].log_data[9].valid := 1, [494].log_data[10].valid := 1, [494].log_data[11].valid := 1, [494].log_data[12].valid := 1, [494].log_data[13].valid := 1, [494].log_data[14].valid := 1, [494].log_data[15].valid := 1, [494].log_data[16].valid := 1, [494].log_data[17].valid := 1, [494].log_data[18].valid := 1, [494].log_data[19].valid := 1, [494].time.Year := 2023, [494].time.Month := 1, [494].time.Day := 12, [494].time.Hour := 19, [494].time.Minute := 59, [494].time.Second := 59, [495].log_data[0].min := 1.0, [495].log_data[0].max := 1.0, [495].log_data[0].total := 900.0, [495].log_data[0].time := 900.0, [495].log_data[0].valid := 1, [495].log_data[1].valid := 1, [495].log_data[2].valid := 1, [495].log_data[3].valid := 1, [495].log_data[4].valid := 1, [495].log_data[5].valid := 1, [495].log_data[6].valid := 1, [495].log_data[7].valid := 1, [495].log_data[8].valid := 1, [495].log_data[9].valid := 1, [495].log_data[10].valid := 1, [495].log_data[11].valid := 1, [495].log_data[12].valid := 1, [495].log_data[13].valid := 1, [495].log_data[14].valid := 1, [495].log_data[15].valid := 1, [495].log_data[16].valid := 1, [495].log_data[17].valid := 1, [495].log_data[18].valid := 1, [495].log_data[19].valid := 1, [495].time.Year := 2023, [495].time.Month := 1, [495].time.Day := 12, [495].time.Hour := 20, [495].time.Minute := 14, [495].time.Second := 59, [496].log_data[0].min := 1.0,
        [496].log_data[0].max := 1.0, [496].log_data[0].total := 900.0, [496].log_data[0].time := 900.0, [496].log_data[0].minminute := 15, [496].log_data[0].maxminute := 15, [496].log_data[0].valid := 1, [496].log_data[1].valid := 1, [496].log_data[2].valid := 1, [496].log_data[3].valid := 1, [496].log_data[4].valid := 1, [496].log_data[5].valid := 1, [496].log_data[6].valid := 1, [496].log_data[7].valid := 1, [496].log_data[8].valid := 1, [496].log_data[9].valid := 1, [496].log_data[10].valid := 1, [496].log_data[11].valid := 1, [496].log_data[12].valid := 1, [496].log_data[13].valid := 1, [496].log_data[14].valid := 1, [496].log_data[15].valid := 1, [496].log_data[16].valid := 1, [496].log_data[17].valid := 1, [496].log_data[18].valid := 1, [496].log_data[19].valid := 1, [496].time.Year := 2023, [496].time.Month := 1, [496].time.Day := 12, [496].time.Hour := 20, [496].time.Minute := 29, [496].time.Second := 59, [497].log_data[0].min := 1.0, [497].log_data[0].max := 1.0, [497].log_data[0].total := 900.0, [497].log_data[0].time := 900.0, [497].log_data[0].minminute := 30, [497].log_data[0].maxminute := 30, [497].log_data[0].valid := 1, [497].log_data[1].valid := 1, [497].log_data[2].valid := 1, [497].log_data[3].valid := 1, [497].log_data[4].valid := 1, [497].log_data[5].valid := 1, [497].log_data[6].valid := 1, [497].log_data[7].valid := 1, [497].log_data[8].valid := 1, [497].log_data[9].valid := 1, [497].log_data[10].valid := 1, [497].log_data[11].valid := 1, [497].log_data[12].valid := 1, [497].log_data[13].valid := 1, [497].log_data[14].valid := 1, [497].log_data[15].valid := 1, [497].log_data[16].valid := 1, [497].log_data[17].valid := 1, [497].log_data[18].valid := 1, [497].log_data[19].valid := 1, [497].time.Year := 2023, [497].time.Month := 1, [497].time.Day := 12,
        [497].time.Hour := 20, [497].time.Minute := 44, [497].time.Second := 59, [498].log_data[0].min := 1.0, [498].log_data[0].max := 1.0, [498].log_data[0].total := 900.0, [498].log_data[0].time := 900.0, [498].log_data[0].minminute := 45, [498].log_data[0].maxminute := 45, [498].log_data[0].valid := 1, [498].log_data[1].valid := 1, [498].log_data[2].valid := 1, [498].log_data[3].valid := 1, [498].log_data[4].valid := 1, [498].log_data[5].valid := 1, [498].log_data[6].valid := 1, [498].log_data[7].valid := 1, [498].log_data[8].valid := 1, [498].log_data[9].valid := 1, [498].log_data[10].valid := 1, [498].log_data[11].valid := 1, [498].log_data[12].valid := 1, [498].log_data[13].valid := 1, [498].log_data[14].valid := 1, [498].log_data[15].valid := 1, [498].log_data[16].valid := 1, [498].log_data[17].valid := 1, [498].log_data[18].valid := 1, [498].log_data[19].valid := 1, [498].time.Year := 2023, [498].time.Month := 1, [498].time.Day := 12, [498].time.Hour := 20, [498].time.Minute := 59, [498].time.Second := 59, [499].log_data[0].min := 1.0, [499].log_data[0].max := 1.0, [499].log_data[0].total := 900.0, [499].log_data[0].time := 900.0, [499].log_data[0].valid := 1, [499].log_data[1].valid := 1, [499].log_data[2].valid := 1, [499].log_data[3].valid := 1, [499].log_data[4].valid := 1, [499].log_data[5].valid := 1, [499].log_data[6].valid := 1, [499].log_data[7].valid := 1, [499].log_data[8].valid := 1, [499].log_data[9].valid := 1, [499].log_data[10].valid := 1, [499].log_data[11].valid := 1, [499].log_data[12].valid := 1, [499].log_data[13].valid := 1, [499].log_data[14].valid := 1, [499].log_data[15].valid := 1, [499].log_data[16].valid := 1, [499].log_data[17].valid := 1, [499].log_data[18].valid := 1, [499].log_data[19].valid := 1, [499].time.Year := 2023,
        [499].time.Month := 1, [499].time.Day := 12, [499].time.Hour := 21, [499].time.Minute := 14, [499].time.Second := 59, [500].log_data[0].min := 1.0, [500].log_data[0].max := 1.0, [500].log_data[0].total := 900.0, [500].log_data[0].time := 900.0, [500].log_data[0].minminute := 15, [500].log_data[0].maxminute := 15, [500].log_data[0].valid := 1, [500].log_data[1].valid := 1, [500].log_data[2].valid := 1, [500].log_data[3].valid := 1, [500].log_data[4].valid := 1, [500].log_data[5].valid := 1, [500].log_data[6].valid := 1, [500].log_data[7].valid := 1, [500].log_data[8].valid := 1, [500].log_data[9].valid := 1, [500].log_data[10].valid := 1, [500].log_data[11].valid := 1, [500].log_data[12].valid := 1, [500].log_data[13].valid := 1, [500].log_data[14].valid := 1, [500].log_data[15].valid := 1, [500].log_data[16].valid := 1, [500].log_data[17].valid := 1, [500].log_data[18].valid := 1, [500].log_data[19].valid := 1, [500].time.Year := 2023, [500].time.Month := 1, [500].time.Day := 12, [500].time.Hour := 21, [500].time.Minute := 29, [500].time.Second := 59, [501].log_data[0].min := 1.0, [501].log_data[0].max := 1.0, [501].log_data[0].total := 900.0, [501].log_data[0].time := 900.0, [501].log_data[0].minminute := 30, [501].log_data[0].maxminute := 30, [501].log_data[0].valid := 1, [501].log_data[1].valid := 1, [501].log_data[2].valid := 1, [501].log_data[3].valid := 1, [501].log_data[4].valid := 1, [501].log_data[5].valid := 1, [501].log_data[6].valid := 1, [501].log_data[7].valid := 1, [501].log_data[8].valid := 1, [501].log_data[9].valid := 1, [501].log_data[10].valid := 1, [501].log_data[11].valid := 1, [501].log_data[12].valid := 1, [501].log_data[13].valid := 1, [501].log_data[14].valid := 1, [501].log_data[15].valid := 1, [501].log_data[16].valid := 1,
        [501].log_data[17].valid := 1, [501].log_data[18].valid := 1, [501].log_data[19].valid := 1, [501].time.Year := 2023, [501].time.Month := 1, [501].time.Day := 12, [501].time.Hour := 21, [501].time.Minute := 44, [501].time.Second := 59, [502].log_data[0].min := 1.0, [502].log_data[0].max := 1.0, [502].log_data[0].total := 900.0, [502].log_data[0].time := 900.0, [502].log_data[0].minminute := 45, [502].log_data[0].maxminute := 45, [502].log_data[0].valid := 1, [502].log_data[1].valid := 1, [502].log_data[2].valid := 1, [502].log_data[3].valid := 1, [502].log_data[4].valid := 1, [502].log_data[5].valid := 1, [502].log_data[6].valid := 1, [502].log_data[7].valid := 1, [502].log_data[8].valid := 1, [502].log_data[9].valid := 1, [502].log_data[10].valid := 1, [502].log_data[11].valid := 1, [502].log_data[12].valid := 1, [502].log_data[13].valid := 1, [502].log_data[14].valid := 1, [502].log_data[15].valid := 1, [502].log_data[16].valid := 1, [502].log_data[17].valid := 1, [502].log_data[18].valid := 1, [502].log_data[19].valid := 1, [502].time.Year := 2023, [502].time.Month := 1, [502].time.Day := 12, [502].time.Hour := 21, [502].time.Minute := 59, [502].time.Second := 59, [503].log_data[0].min := 1.0, [503].log_data[0].max := 1.0, [503].log_data[0].total := 900.0, [503].log_data[0].time := 900.0, [503].log_data[0].valid := 1, [503].log_data[1].valid := 1, [503].log_data[2].valid := 1, [503].log_data[3].valid := 1, [503].log_data[4].valid := 1, [503].log_data[5].valid := 1, [503].log_data[6].valid := 1, [503].log_data[7].valid := 1, [503].log_data[8].valid := 1, [503].log_data[9].valid := 1, [503].log_data[10].valid := 1, [503].log_data[11].valid := 1, [503].log_data[12].valid := 1, [503].log_data[13].valid := 1, [503].log_data[14].valid := 1,
        [503].log_data[15].valid := 1, [503].log_data[16].valid := 1, [503].log_data[17].valid := 1, [503].log_data[18].valid := 1, [503].log_data[19].valid := 1, [503].time.Year := 2023, [503].time.Month := 1, [503].time.Day := 12, [503].time.Hour := 22, [503].time.Minute := 14, [503].time.Second := 59, [504].log_data[0].min := 1.0, [504].log_data[0].max := 1.0, [504].log_data[0].total := 900.0, [504].log_data[0].time := 900.0, [504].log_data[0].minminute := 15, [504].log_data[0].maxminute := 15, [504].log_data[0].valid := 1, [504].log_data[1].valid := 1, [504].log_data[2].valid := 1, [504].log_data[3].valid := 1, [504].log_data[4].valid := 1, [504].log_data[5].valid := 1, [504].log_data[6].valid := 1, [504].log_data[7].valid := 1, [504].log_data[8].valid := 1, [504].log_data[9].valid := 1, [504].log_data[10].valid := 1, [504].log_data[11].valid := 1, [504].log_data[12].valid := 1, [504].log_data[13].valid := 1, [504].log_data[14].valid := 1, [504].log_data[15].valid := 1, [504].log_data[16].valid := 1, [504].log_data[17].valid := 1, [504].log_data[18].valid := 1, [504].log_data[19].valid := 1, [504].time.Year := 2023, [504].time.Month := 1, [504].time.Day := 12, [504].time.Hour := 22, [504].time.Minute := 29, [504].time.Second := 59, [505].log_data[0].min := 1.0, [505].log_data[0].max := 1.0, [505].log_data[0].total := 900.0, [505].log_data[0].time := 900.0, [505].log_data[0].minminute := 30, [505].log_data[0].maxminute := 30, [505].log_data[0].valid := 1, [505].log_data[1].valid := 1, [505].log_data[2].valid := 1, [505].log_data[3].valid := 1, [505].log_data[4].valid := 1, [505].log_data[5].valid := 1, [505].log_data[6].valid := 1, [505].log_data[7].valid := 1, [505].log_data[8].valid := 1, [505].log_data[9].valid := 1, [505].log_data[10].valid := 1,
        [505].log_data[11].valid := 1, [505].log_data[12].valid := 1, [505].log_data[13].valid := 1, [505].log_data[14].valid := 1, [505].log_data[15].valid := 1, [505].log_data[16].valid := 1, [505].log_data[17].valid := 1, [505].log_data[18].valid := 1, [505].log_data[19].valid := 1, [505].time.Year := 2023, [505].time.Month := 1, [505].time.Day := 12, [505].time.Hour := 22, [505].time.Minute := 44, [505].time.Second := 59, [506].log_data[0].min := 1.0, [506].log_data[0].max := 1.0, [506].log_data[0].total := 900.0, [506].log_data[0].time := 900.0, [506].log_data[0].minminute := 45, [506].log_data[0].maxminute := 45, [506].log_data[0].valid := 1, [506].log_data[1].valid := 1, [506].log_data[2].valid := 1, [506].log_data[3].valid := 1, [506].log_data[4].valid := 1, [506].log_data[5].valid := 1, [506].log_data[6].valid := 1, [506].log_data[7].valid := 1, [506].log_data[8].valid := 1, [506].log_data[9].valid := 1, [506].log_data[10].valid := 1, [506].log_data[11].valid := 1, [506].log_data[12].valid := 1, [506].log_data[13].valid := 1, [506].log_data[14].valid := 1, [506].log_data[15].valid := 1, [506].log_data[16].valid := 1, [506].log_data[17].valid := 1, [506].log_data[18].valid := 1, [506].log_data[19].valid := 1, [506].time.Year := 2023, [506].time.Month := 1, [506].time.Day := 12, [506].time.Hour := 22, [506].time.Minute := 59, [506].time.Second := 59, [507].log_data[0].min := 1.0, [507].log_data[0].max := 1.0, [507].log_data[0].total := 900.0, [507].log_data[0].time := 900.0, [507].log_data[0].valid := 1, [507].log_data[1].valid := 1, [507].log_data[2].valid := 1, [507].log_data[3].valid := 1, [507].log_data[4].valid := 1, [507].log_data[5].valid := 1, [507].log_data[6].valid := 1, [507].log_data[7].valid := 1, [507].log_data[8].valid := 1,
        [507].log_data[9].valid := 1, [507].log_data[10].valid := 1, [507].log_data[11].valid := 1, [507].log_data[12].valid := 1, [507].log_data[13].valid := 1, [507].log_data[14].valid := 1, [507].log_data[15].valid := 1, [507].log_data[16].valid := 1, [507].log_data[17].valid := 1, [507].log_data[18].valid := 1, [507].log_data[19].valid := 1, [507].time.Year := 2023, [507].time.Month := 1, [507].time.Day := 12, [507].time.Hour := 23, [507].time.Minute := 14, [507].time.Second := 59, [508].log_data[0].min := 1.0, [508].log_data[0].max := 1.0, [508].log_data[0].total := 900.0, [508].log_data[0].time := 900.0, [508].log_data[0].minminute := 15, [508].log_data[0].maxminute := 15, [508].log_data[0].valid := 1, [508].log_data[1].valid := 1, [508].log_data[2].valid := 1, [508].log_data[3].valid := 1, [508].log_data[4].valid := 1, [508].log_data[5].valid := 1, [508].log_data[6].valid := 1, [508].log_data[7].valid := 1, [508].log_data[8].valid := 1, [508].log_data[9].valid := 1, [508].log_data[10].valid := 1, [508].log_data[11].valid := 1, [508].log_data[12].valid := 1, [508].log_data[13].valid := 1, [508].log_data[14].valid := 1, [508].log_data[15].valid := 1, [508].log_data[16].valid := 1, [508].log_data[17].valid := 1, [508].log_data[18].valid := 1, [508].log_data[19].valid := 1, [508].time.Year := 2023, [508].time.Month := 1, [508].time.Day := 12, [508].time.Hour := 23, [508].time.Minute := 29, [508].time.Second := 59, [509].log_data[0].min := 1.0, [509].log_data[0].max := 1.0, [509].log_data[0].total := 900.0, [509].log_data[0].time := 900.0, [509].log_data[0].minminute := 30, [509].log_data[0].maxminute := 30, [509].log_data[0].valid := 1, [509].log_data[1].valid := 1, [509].log_data[2].valid := 1, [509].log_data[3].valid := 1, [509].log_data[4].valid := 1,
        [509].log_data[5].valid := 1, [509].log_data[6].valid := 1, [509].log_data[7].valid := 1, [509].log_data[8].valid := 1, [509].log_data[9].valid := 1, [509].log_data[10].valid := 1, [509].log_data[11].valid := 1, [509].log_data[12].valid := 1, [509].log_data[13].valid := 1, [509].log_data[14].valid := 1, [509].log_data[15].valid := 1, [509].log_data[16].valid := 1, [509].log_data[17].valid := 1, [509].log_data[18].valid := 1, [509].log_data[19].valid := 1, [509].time.Year := 2023, [509].time.Month := 1, [509].time.Day := 12, [509].time.Hour := 23, [509].time.Minute := 44, [509].time.Second := 59, [510].log_data[0].min := 1.0, [510].log_data[0].max := 1.0, [510].log_data[0].total := 900.0, [510].log_data[0].time := 900.0, [510].log_data[0].minminute := 45, [510].log_data[0].maxminute := 45, [510].log_data[0].valid := 1, [510].log_data[1].valid := 1, [510].log_data[2].valid := 1, [510].log_data[3].valid := 1, [510].log_data[4].valid := 1, [510].log_data[5].valid := 1, [510].log_data[6].valid := 1, [510].log_data[7].valid := 1, [510].log_data[8].valid := 1, [510].log_data[9].valid := 1, [510].log_data[10].valid := 1, [510].log_data[11].valid := 1, [510].log_data[12].valid := 1, [510].log_data[13].valid := 1, [510].log_data[14].valid := 1, [510].log_data[15].valid := 1, [510].log_data[16].valid := 1, [510].log_data[17].valid := 1, [510].log_data[18].valid := 1, [510].log_data[19].valid := 1, [510].time.Year := 2023, [510].time.Month := 1, [510].time.Day := 12, [510].time.Hour := 23, [510].time.Minute := 59, [510].time.Second := 59, [511].log_data[0].min := 1.0, [511].log_data[0].max := 1.0, [511].log_data[0].total := 900.0, [511].log_data[0].time := 900.0, [511].log_data[0].valid := 1, [511].log_data[1].valid := 1, [511].log_data[2].valid := 1,
        [511].log_data[3].valid := 1, [511].log_data[4].valid := 1, [511].log_data[5].valid := 1, [511].log_data[6].valid := 1, [511].log_data[7].valid := 1, [511].log_data[8].valid := 1, [511].log_data[9].valid := 1, [511].log_data[10].valid := 1, [511].log_data[11].valid := 1, [511].log_data[12].valid := 1, [511].log_data[13].valid := 1, [511].log_data[14].valid := 1, [511].log_data[15].valid := 1, [511].log_data[16].valid := 1, [511].log_data[17].valid := 1, [511].log_data[18].valid := 1, [511].log_data[19].valid := 1, [511].time.Year := 2023, [511].time.Month := 1, [511].time.Day := 13, [511].time.Minute := 14, [511].time.Second := 59, [512].log_data[0].min := 1.0, [512].log_data[0].max := 1.0, [512].log_data[0].total := 900.0, [512].log_data[0].time := 900.0, [512].log_data[0].minminute := 15, [512].log_data[0].maxminute := 15, [512].log_data[0].valid := 1, [512].log_data[1].valid := 1, [512].log_data[2].valid := 1, [512].log_data[3].valid := 1, [512].log_data[4].valid := 1, [512].log_data[5].valid := 1, [512].log_data[6].valid := 1, [512].log_data[7].valid := 1, [512].log_data[8].valid := 1, [512].log_data[9].valid := 1, [512].log_data[10].valid := 1, [512].log_data[11].valid := 1, [512].log_data[12].valid := 1, [512].log_data[13].valid := 1, [512].log_data[14].valid := 1, [512].log_data[15].valid := 1, [512].log_data[16].valid := 1, [512].log_data[17].valid := 1, [512].log_data[18].valid := 1, [512].log_data[19].valid := 1, [512].time.Year := 2023, [512].time.Month := 1, [512].time.Day := 13, [512].time.Minute := 29, [512].time.Second := 59, [513].log_data[0].min := 1.0, [513].log_data[0].max := 1.0, [513].log_data[0].total := 900.0, [513].log_data[0].time := 900.0, [513].log_data[0].minminute := 30, [513].log_data[0].maxminute := 30, [513].log_data[0].valid := 1,
        [513].log_data[1].valid := 1, [513].log_data[2].valid := 1, [513].log_data[3].valid := 1, [513].log_data[4].valid := 1, [513].log_data[5].valid := 1, [513].log_data[6].valid := 1, [513].log_data[7].valid := 1, [513].log_data[8].valid := 1, [513].log_data[9].valid := 1, [513].log_data[10].valid := 1, [513].log_data[11].valid := 1, [513].log_data[12].valid := 1, [513].log_data[13].valid := 1, [513].log_data[14].valid := 1, [513].log_data[15].valid := 1, [513].log_data[16].valid := 1, [513].log_data[17].valid := 1, [513].log_data[18].valid := 1, [513].log_data[19].valid := 1, [513].time.Year := 2023, [513].time.Month := 1, [513].time.Day := 13, [513].time.Minute := 44, [513].time.Second := 59, [514].log_data[0].min := 1.0, [514].log_data[0].max := 1.0, [514].log_data[0].total := 900.0, [514].log_data[0].time := 900.0, [514].log_data[0].minminute := 45, [514].log_data[0].maxminute := 45, [514].log_data[0].valid := 1, [514].log_data[1].valid := 1, [514].log_data[2].valid := 1, [514].log_data[3].valid := 1, [514].log_data[4].valid := 1, [514].log_data[5].valid := 1, [514].log_data[6].valid := 1, [514].log_data[7].valid := 1, [514].log_data[8].valid := 1, [514].log_data[9].valid := 1, [514].log_data[10].valid := 1, [514].log_data[11].valid := 1, [514].log_data[12].valid := 1, [514].log_data[13].valid := 1, [514].log_data[14].valid := 1, [514].log_data[15].valid := 1, [514].log_data[16].valid := 1, [514].log_data[17].valid := 1, [514].log_data[18].valid := 1, [514].log_data[19].valid := 1, [514].time.Year := 2023, [514].time.Month := 1, [514].time.Day := 13, [514].time.Minute := 59, [514].time.Second := 59, [515].log_data[0].min := 1.0, [515].log_data[0].max := 1.0, [515].log_data[0].total := 899.5, [515].log_data[0].time := 899.5, [515].log_data[0].valid := 1,
        [515].log_data[1].valid := 1, [515].log_data[2].valid := 1, [515].log_data[3].valid := 1, [515].log_data[4].valid := 1, [515].log_data[5].valid := 1, [515].log_data[6].valid := 1, [515].log_data[7].valid := 1, [515].log_data[8].valid := 1, [515].log_data[9].valid := 1, [515].log_data[10].valid := 1, [515].log_data[11].valid := 1, [515].log_data[12].valid := 1, [515].log_data[13].valid := 1, [515].log_data[14].valid := 1, [515].log_data[15].valid := 1, [515].log_data[16].valid := 1, [515].log_data[17].valid := 1, [515].log_data[18].valid := 1, [515].log_data[19].valid := 1, [515].time.Year := 2023, [515].time.Month := 1, [515].time.Day := 13, [515].time.Hour := 1, [515].time.Minute := 14, [515].time.Second := 59, [516].log_data[0].min := 1.0, [516].log_data[0].max := 1.0, [516].log_data[0].total := 900.0, [516].log_data[0].time := 900.0, [516].log_data[0].minminute := 15, [516].log_data[0].maxminute := 15, [516].log_data[0].valid := 1, [516].log_data[1].valid := 1, [516].log_data[2].valid := 1, [516].log_data[3].valid := 1, [516].log_data[4].valid := 1, [516].log_data[5].valid := 1, [516].log_data[6].valid := 1, [516].log_data[7].valid := 1, [516].log_data[8].valid := 1, [516].log_data[9].valid := 1, [516].log_data[10].valid := 1, [516].log_data[11].valid := 1, [516].log_data[12].valid := 1, [516].log_data[13].valid := 1, [516].log_data[14].valid := 1, [516].log_data[15].valid := 1, [516].log_data[16].valid := 1, [516].log_data[17].valid := 1, [516].log_data[18].valid := 1, [516].log_data[19].valid := 1, [516].time.Year := 2023, [516].time.Month := 1, [516].time.Day := 13, [516].time.Hour := 1, [516].time.Minute := 29, [516].time.Second := 59, [517].log_data[0].min := 1.0, [517].log_data[0].max := 1.0, [517].log_data[0].total := 900.0,
        [517].log_data[0].time := 900.0, [517].log_data[0].minminute := 30, [517].log_data[0].maxminute := 30, [517].log_data[0].valid := 1, [517].log_data[1].valid := 1, [517].log_data[2].valid := 1, [517].log_data[3].valid := 1, [517].log_data[4].valid := 1, [517].log_data[5].valid := 1, [517].log_data[6].valid := 1, [517].log_data[7].valid := 1, [517].log_data[8].valid := 1, [517].log_data[9].valid := 1, [517].log_data[10].valid := 1, [517].log_data[11].valid := 1, [517].log_data[12].valid := 1, [517].log_data[13].valid := 1, [517].log_data[14].valid := 1, [517].log_data[15].valid := 1, [517].log_data[16].valid := 1, [517].log_data[17].valid := 1, [517].log_data[18].valid := 1, [517].log_data[19].valid := 1, [517].time.Year := 2023, [517].time.Month := 1, [517].time.Day := 13, [517].time.Hour := 1, [517].time.Minute := 44, [517].time.Second := 59, [518].log_data[0].min := 1.0, [518].log_data[0].max := 1.0, [518].log_data[0].total := 900.0, [518].log_data[0].time := 900.0, [518].log_data[0].minminute := 45, [518].log_data[0].maxminute := 45, [518].log_data[0].valid := 1, [518].log_data[1].valid := 1, [518].log_data[2].valid := 1, [518].log_data[3].valid := 1, [518].log_data[4].valid := 1, [518].log_data[5].valid := 1, [518].log_data[6].valid := 1, [518].log_data[7].valid := 1, [518].log_data[8].valid := 1, [518].log_data[9].valid := 1, [518].log_data[10].valid := 1, [518].log_data[11].valid := 1, [518].log_data[12].valid := 1, [518].log_data[13].valid := 1, [518].log_data[14].valid := 1, [518].log_data[15].valid := 1, [518].log_data[16].valid := 1, [518].log_data[17].valid := 1, [518].log_data[18].valid := 1, [518].log_data[19].valid := 1, [518].time.Year := 2023, [518].time.Month := 1, [518].time.Day := 13, [518].time.Hour := 1, [518].time.Minute := 59,
        [518].time.Second := 59, [519].log_data[0].min := 1.0, [519].log_data[0].max := 1.0, [519].log_data[0].total := 900.0, [519].log_data[0].time := 900.0, [519].log_data[0].valid := 1, [519].log_data[1].valid := 1, [519].log_data[2].valid := 1, [519].log_data[3].valid := 1, [519].log_data[4].valid := 1, [519].log_data[5].valid := 1, [519].log_data[6].valid := 1, [519].log_data[7].valid := 1, [519].log_data[8].valid := 1, [519].log_data[9].valid := 1, [519].log_data[10].valid := 1, [519].log_data[11].valid := 1, [519].log_data[12].valid := 1, [519].log_data[13].valid := 1, [519].log_data[14].valid := 1, [519].log_data[15].valid := 1, [519].log_data[16].valid := 1, [519].log_data[17].valid := 1, [519].log_data[18].valid := 1, [519].log_data[19].valid := 1, [519].time.Year := 2023, [519].time.Month := 1, [519].time.Day := 13, [519].time.Hour := 2, [519].time.Minute := 14, [519].time.Second := 59, [520].log_data[0].min := 1.0, [520].log_data[0].max := 1.0, [520].log_data[0].total := 900.0, [520].log_data[0].time := 900.0, [520].log_data[0].minminute := 15, [520].log_data[0].maxminute := 15, [520].log_data[0].valid := 1, [520].log_data[1].valid := 1, [520].log_data[2].valid := 1, [520].log_data[3].valid := 1, [520].log_data[4].valid := 1, [520].log_data[5].valid := 1, [520].log_data[6].valid := 1, [520].log_data[7].valid := 1, [520].log_data[8].valid := 1, [520].log_data[9].valid := 1, [520].log_data[10].valid := 1, [520].log_data[11].valid := 1, [520].log_data[12].valid := 1, [520].log_data[13].valid := 1, [520].log_data[14].valid := 1, [520].log_data[15].valid := 1, [520].log_data[16].valid := 1, [520].log_data[17].valid := 1, [520].log_data[18].valid := 1, [520].log_data[19].valid := 1, [520].time.Year := 2023, [520].time.Month := 1, [520].time.Day := 13,
